LIN {X 0,Y 373.516,Z 952.695,A -85,B 0,C 180,E1 18425.825,E2 18425.825} C_VEL
LIN {X 0,Y 376.652,Z 940.388,A -85,B 0,C 180,E1 18422.322,E2 18422.322} C_VEL
LIN {X 0,Y 380.104,Z 927.885,A -85,B 0,C 180,E1 18419.319,E2 18419.319} C_VEL
LIN {X 0,Y 384.269,Z 913.225,A -85,B 0,C 180,E1 18416.347,E2 18416.347} C_VEL
LIN {X 0,Y 388.82,Z 897.706,A -85,B 0,C 180,E1 18413.653,E2 18413.653} C_VEL
LIN {X 0,Y 393.494,Z 881.198,A -85,B 0,C 180,E1 18411.233,E2 18411.233} C_VEL
LIN {X 0,Y 398.594,Z 862.696,A -85,B 0,C 180,E1 18408.917,E2 18408.917} C_VEL
LIN {X 0,Y 403.277,Z 844.718,A -85,B 0,C 180,E1 18407.02,E2 18407.02} C_VEL
LIN {X 0,Y 408.104,Z 824.554,A -85,B 0,C 180,E1 18405.227,E2 18405.227} C_VEL
LIN {X 0,Y 411.988,Z 806.631,A -85,B 0,C 180,E1 18403.886,E2 18403.886} C_VEL
LIN {X 0,Y 416.257,Z 784.1,A -85,B 0,C 180,E1 18402.494,E2 18402.494} C_VEL
LIN {X 0,Y 419.472,Z 764.172,A -85,B 0,C 180,E1 18401.502,E2 18401.502} C_VEL
LIN {X 0,Y 422.462,Z 740.832,A -85,B 0,C 180,E1 18400.598,E2 18400.598} C_VEL
LIN {X 0,Y 424.7,Z 718.024,A -85,B 0,C 180,E1 18399.95,E2 18399.95} C_VEL
LIN {X 0,Y 427.255,Z 666.6,A -85,B 0,C 180,E1 18398.953,E2 18398.953} C_VEL
LIN {X 0,Y 436.486,Z 468.995,A -85,B 0,C 180,E1 18395.218,E2 18395.218} C_VEL
LIN {X 0,Y 426.222,Z 453.887,A -85,B 0,C 180,E1 18392.733,E2 18392.733} C_VEL
LIN {X 0,Y 415.395,Z 439.157,A -85,B 0,C 180,E1 18389.805,E2 18389.805} C_VEL
LIN {X 0,Y 406.554,Z 427.967,A -85,B 0,C 180,E1 18387.103,E2 18387.103} C_VEL
LIN {X 0,Y 401.998,Z 422.413,A -85,B 0,C 180,E1 18385.565,E2 18385.565} C_VEL
LIN {X 0,Y 398.336,Z 417.839,A -85,B 0,C 180,E1 18384.23,E2 18384.23} C_VEL
LIN {X 0,Y 393.924,Z 412.857,A -85,B 0,C 180,E1 18382.511,E2 18382.511} C_VEL
LIN {X 0,Y 392.689,Z 411.071,A -85,B 0,C 180,E1 18381.981,E2 18381.981} C_VEL
LIN {X 0,Y 389.373,Z 407.904,A -85,B 0,C 180,E1 18380.558,E2 18380.558} C_VEL
LIN {X 0,Y 387.428,Z 404.914,A -85,B 0,C 180,E1 18379.603,E2 18379.603} C_VEL
LIN {X 0,Y 383.951,Z 402.051,A -85,B 0,C 180,E1 18377.896,E2 18377.896} C_VEL
LIN {X 0,Y 382.021,Z 398.482,A -85,B 0,C 180,E1 18376.733,E2 18376.733} C_VEL
LIN {X 0,Y 378.538,Z 396.352,A -85,B 0,C 180,E1 18374.689,E2 18374.689} C_VEL
LIN {X 0,Y 376.63,Z 393.429,A -85,B 0,C 180,E1 18373.276,E2 18373.276} C_VEL
LIN {X 0,Y 376.047,Z 391.834,A -85,B 0,C 180,E1 18372.75,E2 18372.75} C_VEL
LIN {X 0,Y 372.15,Z 389.796,A -85,B 0,C 180,E1 18369.433,E2 18369.433} C_VEL
LIN {X 0,Y 370.046,Z 386.524,A -85,B 0,C 180,E1 18366.594,E2 18366.594} C_VEL
LIN {X 0,Y 369.697,Z 384.985,A -85,B 0,C 180,E1 18365.639,E2 18365.639} C_VEL
LIN {X 0,Y 369.684,Z 384.983,A -85,B 0,C 180,E1 18361.705,E2 18361.705} C_VEL
LIN {X 0,Y 369.678,Z 384.981,A -85,B 0,C 180,E1 18357.675,E2 18357.675} C_VEL
LIN {X 0,Y 369.728,Z 385.142,A -85,B 0,C 180,E1 18354.608,E2 18354.608} C_VEL
LIN {X 0,Y 370.458,Z 387.543,A -85,B 0,C 180,E1 18353.18,E2 18353.18} C_VEL
LIN {X 0,Y 373.077,Z 390.581,A -85,B 0,C 180,E1 18350.124,E2 18350.124} C_VEL
LIN {X 0,Y 376.149,Z 392.051,A -85,B 0,C 180,E1 18347.645,E2 18347.645} C_VEL
LIN {X 0,Y 377.796,Z 395.551,A -85,B 0,C 180,E1 18346.299,E2 18346.299} C_VEL
LIN {X 0,Y 380.714,Z 397.973,A -85,B 0,C 180,E1 18344.462,E2 18344.462} C_VEL
LIN {X 0,Y 382.155,Z 398.748,A -85,B 0,C 180,E1 18343.665,E2 18343.665} C_VEL
LIN {X 0,Y 384.237,Z 402.413,A -85,B 0,C 180,E1 18342.431,E2 18342.431} C_VEL
LIN {X 0,Y 387.814,Z 405.39,A -85,B 0,C 180,E1 18340.692,E2 18340.692} C_VEL
LIN {X 0,Y 390.392,Z 409.19,A -85,B 0,C 180,E1 18339.459,E2 18339.459} C_VEL
LIN {X 0,Y 393.289,Z 411.748,A -85,B 0,C 180,E1 18338.252,E2 18338.252} C_VEL
LIN {X 0,Y 396.375,Z 415.904,A -85,B 0,C 180,E1 18336.984,E2 18336.984} C_VEL
LIN {X 0,Y 398.445,Z 418.003,A -85,B 0,C 180,E1 18336.21,E2 18336.21} C_VEL
LIN {X 0,Y 405.924,Z 427.773,A -85,B 0,C 180,E1 18333.563,E2 18333.563} C_VEL
LIN {X 0,Y 413.865,Z 438.738,A -85,B 0,C 180,E1 18331.068,E2 18331.068} C_VEL
LIN {X 0,Y 422.741,Z 451.748,A -85,B 0,C 180,E1 18328.566,E2 18328.566} C_VEL
LIN {X 0,Y 431.121,Z 464.861,A -85,B 0,C 180,E1 18326.418,E2 18326.418} C_VEL
LIN {X 0,Y 436.61,Z 474.131,A -85,B 0,C 180,E1 18325.098,E2 18325.098} C_VEL
LIN {X 0,Y 427.077,Z 679.523,A -85,B 0,C 180,E1 18321.22,E2 18321.22} C_VEL
LIN {X 0,Y 424.258,Z 738.023,A -85,B 0,C 180,E1 18320.092,E2 18320.092} C_VEL
LIN {X 0,Y 421.886,Z 761.213,A -85,B 0,C 180,E1 18319.459,E2 18319.459} C_VEL
LIN {X 0,Y 418.914,Z 783.591,A -85,B 0,C 180,E1 18318.636,E2 18318.636} C_VEL
LIN {X 0,Y 415.436,Z 804.583,A -85,B 0,C 180,E1 18317.629,E2 18317.629} C_VEL
LIN {X 0,Y 411.179,Z 826.892,A -85,B 0,C 180,E1 18316.297,E2 18316.297} C_VEL
LIN {X 0,Y 406.878,Z 846.732,A -85,B 0,C 180,E1 18314.845,E2 18314.845} C_VEL
LIN {X 0,Y 401.839,Z 867.94,A -85,B 0,C 180,E1 18312.976,E2 18312.976} C_VEL
LIN {X 0,Y 397.191,Z 886.217,A -85,B 0,C 180,E1 18311.068,E2 18311.068} C_VEL
LIN {X 0,Y 392.279,Z 904.4,A -85,B 0,C 180,E1 18308.825,E2 18308.825} C_VEL
LIN {X 0,Y 387.533,Z 921.911,A -85,B 0,C 180,E1 18306.303,E2 18306.303} C_VEL
LIN {X 0,Y 383.114,Z 937.825,A -85,B 0,C 180,E1 18303.589,E2 18303.589} C_VEL
LIN {X 0,Y 379.106,Z 952.905,A -85,B 0,C 180,E1 18300.595,E2 18300.595} C_VEL
LIN {X 0,Y 375.901,Z 965.517,A -85,B 0,C 180,E1 18297.658,E2 18297.658} C_VEL
LIN {X 0,Y 372.991,Z 978.095,A -85,B 0,C 180,E1 18294.211,E2 18294.211} C_VEL
LIN {X 0,Y 371.011,Z 987.984,A -85,B 0,C 180,E1 18291.002,E2 18291.002} C_VEL
LIN {X 0,Y 369.511,Z 996.933,A -85,B 0,C 180,E1 18287.477,E2 18287.477} C_VEL
LIN {X 0,Y 368.666,Z 1003.581,A -85,B 0,C 180,E1 18284.287,E2 18284.287} C_VEL
LIN {X 0,Y 368.17,Z 1009.216,A -85,B 0,C 180,E1 18280.799,E2 18280.799} C_VEL
LIN {X 0,Y 367.983,Z 1012.808,A -85,B 0,C 180,E1 18277.808,E2 18277.808} C_VEL
LIN {X 0,Y 367.925,Z 1015.554,A -85,B 0,C 180,E1 18274.364,E2 18274.364} C_VEL
LIN {X 0,Y 367.923,Z 1016.636,A -85,B 0,C 180,E1 18271.246,E2 18271.246} C_VEL
LIN {X 0,Y 367.927,Z 1016.566,A -85,B 0,C 180,E1 18268.288,E2 18268.288} C_VEL
LIN {X 0,Y 367.929,Z 1015.054,A -85,B 0,C 180,E1 18264.856,E2 18264.856} C_VEL
LIN {X 0,Y 368.017,Z 1012.314,A -85,B 0,C 180,E1 18261.722,E2 18261.722} C_VEL
LIN {X 0,Y 368.261,Z 1007.893,A -85,B 0,C 180,E1 18258.252,E2 18258.252} C_VEL
LIN {X 0,Y 368.84,Z 1002.025,A -85,B 0,C 180,E1 18254.918,E2 18254.918} C_VEL
LIN {X 0,Y 369.87,Z 994.748,A -85,B 0,C 180,E1 18251.564,E2 18251.564} C_VEL
LIN {X 0,Y 371.459,Z 985.641,A -85,B 0,C 180,E1 18248.198,E2 18248.198} C_VEL
LIN {X 0,Y 373.742,Z 974.864,A -85,B 0,C 180,E1 18244.83,E2 18244.83} C_VEL
LIN {X 0,Y 376.621,Z 962.624,A -85,B 0,C 180,E1 18241.631,E2 18241.631} C_VEL
LIN {X 0,Y 380.349,Z 948.091,A -85,B 0,C 180,E1 18238.399,E2 18238.399} C_VEL
LIN {X 0,Y 384.315,Z 933.523,A -85,B 0,C 180,E1 18235.633,E2 18235.633} C_VEL
LIN {X 0,Y 388.884,Z 916.777,A -85,B 0,C 180,E1 18232.926,E2 18232.926} C_VEL
LIN {X 0,Y 393.604,Z 899.717,A -85,B 0,C 180,E1 18230.555,E2 18230.555} C_VEL
LIN {X 0,Y 398.399,Z 881.4,A -85,B 0,C 180,E1 18228.407,E2 18228.407} C_VEL
LIN {X 0,Y 403.332,Z 861.809,A -85,B 0,C 180,E1 18226.443,E2 18226.443} C_VEL
LIN {X 0,Y 407.884,Z 842.145,A -85,B 0,C 180,E1 18224.8,E2 18224.8} C_VEL
LIN {X 0,Y 412.556,Z 819.977,A -85,B 0,C 180,E1 18223.265,E2 18223.265} C_VEL
LIN {X 0,Y 416.124,Z 800.624,A -85,B 0,C 180,E1 18222.169,E2 18222.169} C_VEL
LIN {X 0,Y 419.768,Z 777.421,A -85,B 0,C 180,E1 18221.121,E2 18221.121} C_VEL
LIN {X 0,Y 422.274,Z 757.737,A -85,B 0,C 180,E1 18220.438,E2 18220.438} C_VEL
LIN {X 0,Y 424.553,Z 732.637,A -85,B 0,C 180,E1 18219.8,E2 18219.8} C_VEL
LIN {X 0,Y 433.641,Z 535.185,A -85,B 0,C 180,E1 18216.062,E2 18216.062} C_VEL
LIN {X 0,Y 436.481,Z 473.671,A -85,B 0,C 180,E1 18214.879,E2 18214.879} C_VEL
LIN {X 0,Y 426.008,Z 456.76,A -85,B 0,C 180,E1 18212.312,E2 18212.312} C_VEL
LIN {X 0,Y 415.5,Z 441.08,A -85,B 0,C 180,E1 18209.439,E2 18209.439} C_VEL
LIN {X 0,Y 407.607,Z 430.178,A -85,B 0,C 180,E1 18207.027,E2 18207.027} C_VEL
LIN {X 0,Y 403.606,Z 424.766,A -85,B 0,C 180,E1 18205.691,E2 18205.691} C_VEL
LIN {X 0,Y 397.54,Z 416.927,A -85,B 0,C 180,E1 18203.493,E2 18203.493} C_VEL
LIN {X 0,Y 394.055,Z 413.056,A -85,B 0,C 180,E1 18202.135,E2 18202.135} C_VEL
LIN {X 0,Y 392.767,Z 411.133,A -85,B 0,C 180,E1 18201.583,E2 18201.583} C_VEL
LIN {X 0,Y 389.194,Z 407.75,A -85,B 0,C 180,E1 18200.057,E2 18200.057} C_VEL
LIN {X 0,Y 387.321,Z 404.835,A -85,B 0,C 180,E1 18199.138,E2 18199.138} C_VEL
LIN {X 0,Y 384.105,Z 402.262,A -85,B 0,C 180,E1 18197.575,E2 18197.575} C_VEL
LIN {X 0,Y 381.889,Z 398.463,A -85,B 0,C 180,E1 18196.269,E2 18196.269} C_VEL
LIN {X 0,Y 378.287,Z 396.166,A -85,B 0,C 180,E1 18194.151,E2 18194.151} C_VEL
LIN {X 0,Y 376.466,Z 393.014,A -85,B 0,C 180,E1 18192.774,E2 18192.774} C_VEL
LIN {X 0,Y 376.101,Z 391.867,A -85,B 0,C 180,E1 18192.435,E2 18192.435} C_VEL
LIN {X 0,Y 372.429,Z 390.055,A -85,B 0,C 180,E1 18189.425,E2 18189.425} C_VEL
LIN {X 0,Y 370.155,Z 386.892,A -85,B 0,C 180,E1 18186.606,E2 18186.606} C_VEL
LIN {X 0,Y 369.687,Z 384.981,A -85,B 0,C 180,E1 18185.587,E2 18185.587} C_VEL
LIN {X 0,Y 369.689,Z 384.981,A -85,B 0,C 180,E1 18181.549,E2 18181.549} C_VEL
LIN {X 0,Y 369.681,Z 384.984,A -85,B 0,C 180,E1 18177.675,E2 18177.675} C_VEL
LIN {X 0,Y 369.686,Z 385.014,A -85,B 0,C 180,E1 18173.789,E2 18173.789} C_VEL
LIN {X 0,Y 370.975,Z 388.444,A -85,B 0,C 180,E1 18171.631,E2 18171.631} C_VEL
LIN {X 0,Y 374.173,Z 391.196,A -85,B 0,C 180,E1 18168.439,E2 18168.439} C_VEL
LIN {X 0,Y 376.158,Z 392.014,A -85,B 0,C 180,E1 18166.942,E2 18166.942} C_VEL
LIN {X 0,Y 377.412,Z 395.001,A -85,B 0,C 180,E1 18165.893,E2 18165.893} C_VEL
LIN {X 0,Y 380.397,Z 397.79,A -85,B 0,C 180,E1 18163.979,E2 18163.979} C_VEL
LIN {X 0,Y 382.105,Z 398.687,A -85,B 0,C 180,E1 18163.036,E2 18163.036} C_VEL
LIN {X 0,Y 384.066,Z 402.206,A -85,B 0,C 180,E1 18161.874,E2 18161.874} C_VEL
LIN {X 0,Y 387.875,Z 405.412,A -85,B 0,C 180,E1 18160.028,E2 18160.028} C_VEL
LIN {X 0,Y 390.547,Z 409.351,A -85,B 0,C 180,E1 18158.761,E2 18158.761} C_VEL
LIN {X 0,Y 393.213,Z 411.691,A -85,B 0,C 180,E1 18157.657,E2 18157.657} C_VEL
LIN {X 0,Y 396.4,Z 415.938,A -85,B 0,C 180,E1 18156.356,E2 18156.356} C_VEL
LIN {X 0,Y 398.299,Z 417.824,A -85,B 0,C 180,E1 18155.649,E2 18155.649} C_VEL
LIN {X 0,Y 401.875,Z 422.318,A -85,B 0,C 180,E1 18154.347,E2 18154.347} C_VEL
LIN {X 0,Y 403.594,Z 424.397,A -85,B 0,C 180,E1 18153.755,E2 18153.755} C_VEL
LIN {X 0,Y 408.142,Z 430.056,A -85,B 0,C 180,E1 18152.26,E2 18152.26} C_VEL
LIN {X 0,Y 413.122,Z 436.484,A -85,B 0,C 180,E1 18150.732,E2 18150.732} C_VEL
LIN {X 0,Y 419.587,Z 444.835,A -85,B 0,C 180,E1 18148.902,E2 18148.902} C_VEL
LIN {X 0,Y 429.926,Z 459.317,A -85,B 0,C 180,E1 18146.232,E2 18146.232} C_VEL
LIN {X 0,Y 436.465,Z 469.171,A -85,B 0,C 180,E1 18144.678,E2 18144.678} C_VEL
LIN {X 0,Y 426.653,Z 679.212,A -85,B 0,C 180,E1 18140.716,E2 18140.716} C_VEL
LIN {X 0,Y 424.59,Z 718.849,A -85,B 0,C 180,E1 18139.935,E2 18139.935} C_VEL
LIN {X 0,Y 422.399,Z 741.121,A -85,B 0,C 180,E1 18139.298,E2 18139.298} C_VEL
LIN {X 0,Y 419.325,Z 764.94,A -85,B 0,C 180,E1 18138.368,E2 18138.368} C_VEL
LIN {X 0,Y 416.219,Z 784.161,A -85,B 0,C 180,E1 18137.408,E2 18137.408} C_VEL
LIN {X 0,Y 411.978,Z 806.574,A -85,B 0,C 180,E1 18136.024,E2 18136.024} C_VEL
LIN {X 0,Y 408.075,Z 824.581,A -85,B 0,C 180,E1 18134.677,E2 18134.677} C_VEL
LIN {X 0,Y 403.062,Z 845.452,A -85,B 0,C 180,E1 18132.814,E2 18132.814} C_VEL
LIN {X 0,Y 398.238,Z 864.016,A -85,B 0,C 180,E1 18130.841,E2 18130.841} C_VEL
LIN {X 0,Y 393.344,Z 881.688,A -85,B 0,C 180,E1 18128.606,E2 18128.606} C_VEL
LIN {X 0,Y 388.676,Z 898.193,A -85,B 0,C 180,E1 18126.179,E2 18126.179} C_VEL
LIN {X 0,Y 384.149,Z 913.628,A -85,B 0,C 180,E1 18123.485,E2 18123.485} C_VEL
LIN {X 0,Y 380.002,Z 928.214,A -85,B 0,C 180,E1 18120.514,E2 18120.514} C_VEL
LIN {X 0,Y 378.162,Z 934.959,A -85,B 0,C 180,E1 18118.963,E2 18118.963} C_VEL
LIN {X 0,Y 376.147,Z 939.177,A -85,B 0,C 180,E1 18118.021,E2 18118.021} C_VEL
LIN {X 0,Y 367.506,Z 949.935,A -85,B 0,C 180,E1 18115.527,E2 18115.527} C_VEL
LIN {X 0,Y 366.002,Z 952.956,A -85,B 0,C 180,E1 18114.63,E2 18114.63} C_VEL
LIN {X 0,Y 363.682,Z 962.63,A -85,B 0,C 180,E1 18111.276,E2 18111.276} C_VEL
LIN {X 0,Y 362.005,Z 970.702,A -85,B 0,C 180,E1 18107.851,E2 18107.851} C_VEL
LIN {X 0,Y 360.935,Z 977.299,A -85,B 0,C 180,E1 18104.435,E2 18104.435} C_VEL
LIN {X 0,Y 360.306,Z 982.537,A -85,B 0,C 180,E1 18100.875,E2 18100.875} C_VEL
LIN {X 0,Y 360.034,Z 986.031,A -85,B 0,C 180,E1 18097.659,E2 18097.659} C_VEL
LIN {X 0,Y 359.946,Z 988.516,A -85,B 0,C 180,E1 18093.981,E2 18093.981} C_VEL
LIN {X 0,Y 359.922,Z 989.386,A -85,B 0,C 180,E1 18090.954,E2 18090.954} C_VEL
LIN {X 0,Y 359.937,Z 989.147,A -85,B 0,C 180,E1 18087.452,E2 18087.452} C_VEL
LIN {X 0,Y 359.975,Z 987.462,A -85,B 0,C 180,E1 18084.102,E2 18084.102} C_VEL
LIN {X 0,Y 360.165,Z 984.418,A -85,B 0,C 180,E1 18080.574,E2 18080.574} C_VEL
LIN {X 0,Y 360.615,Z 979.736,A -85,B 0,C 180,E1 18077.023,E2 18077.023} C_VEL
LIN {X 0,Y 361.527,Z 973.629,A -85,B 0,C 180,E1 18073.451,E2 18073.451} C_VEL
LIN {X 0,Y 363.012,Z 965.68,A -85,B 0,C 180,E1 18069.863,E2 18069.863} C_VEL
LIN {X 0,Y 365.253,Z 956.02,A -85,B 0,C 180,E1 18066.274,E2 18066.274} C_VEL
LIN {X 0,Y 367.859,Z 945.995,A -85,B 0,C 180,E1 18063.182,E2 18063.182} C_VEL
LIN {X 0,Y 371.648,Z 932.713,A -85,B 0,C 180,E1 18059.723,E2 18059.723} C_VEL
LIN {X 0,Y 375.474,Z 919.99,A -85,B 0,C 180,E1 18056.918,E2 18056.918} C_VEL
LIN {X 0,Y 380.055,Z 904.898,A -85,B 0,C 180,E1 18054.083,E2 18054.083} C_VEL
LIN {X 0,Y 384.914,Z 889.023,A -85,B 0,C 180,E1 18051.533,E2 18051.533} C_VEL
LIN {X 0,Y 389.998,Z 871.654,A -85,B 0,C 180,E1 18049.18,E2 18049.18} C_VEL
LIN {X 0,Y 395.062,Z 853.737,A -85,B 0,C 180,E1 18047.099,E2 18047.099} C_VEL
LIN {X 0,Y 400.045,Z 834.352,A -85,B 0,C 180,E1 18045.22,E2 18045.22} C_VEL
LIN {X 0,Y 404.945,Z 813.698,A -85,B 0,C 180,E1 18043.542,E2 18043.542} C_VEL
LIN {X 0,Y 408.969,Z 794.385,A -85,B 0,C 180,E1 18042.247,E2 18042.247} C_VEL
LIN {X 0,Y 412.949,Z 772.361,A -85,B 0,C 180,E1 18041.039,E2 18041.039} C_VEL
LIN {X 0,Y 415.872,Z 752.629,A -85,B 0,C 180,E1 18040.18,E2 18040.18} C_VEL
LIN {X 0,Y 418.6,Z 729.318,A -85,B 0,C 180,E1 18039.403,E2 18039.403} C_VEL
LIN {X 0,Y 420.287,Z 707.78,A -85,B 0,C 180,E1 18038.891,E2 18038.891} C_VEL
LIN {X 0,Y 430.38,Z 500.127,A -85,B 0,C 180,E1 18034.943,E2 18034.943} C_VEL
LIN {X 0,Y 431.677,Z 473.073,A -85,B 0,C 180,E1 18034.413,E2 18034.413} C_VEL
LIN {X 0,Y 422.102,Z 459.129,A -85,B 0,C 180,E1 18032.01,E2 18032.01} C_VEL
LIN {X 0,Y 412.697,Z 446.062,A -85,B 0,C 180,E1 18029.381,E2 18029.381} C_VEL
LIN {X 0,Y 404.001,Z 434.917,A -85,B 0,C 180,E1 18026.653,E2 18026.653} C_VEL
LIN {X 0,Y 399.715,Z 429.598,A -85,B 0,C 180,E1 18025.166,E2 18025.166} C_VEL
LIN {X 0,Y 395.232,Z 424.08,A -85,B 0,C 180,E1 18023.481,E2 18023.481} C_VEL
LIN {X 0,Y 391.692,Z 419.829,A -85,B 0,C 180,E1 18022.04,E2 18022.04} C_VEL
LIN {X 0,Y 390.567,Z 418.418,A -85,B 0,C 180,E1 18021.553,E2 18021.553} C_VEL
LIN {X 0,Y 387.275,Z 414.949,A -85,B 0,C 180,E1 18020.083,E2 18020.083} C_VEL
LIN {X 0,Y 385.875,Z 412.632,A -85,B 0,C 180,E1 18019.37,E2 18019.37} C_VEL
LIN {X 0,Y 382.317,Z 409.595,A -85,B 0,C 180,E1 18017.582,E2 18017.582} C_VEL
LIN {X 0,Y 380.274,Z 406.175,A -85,B 0,C 180,E1 18016.34,E2 18016.34} C_VEL
LIN {X 0,Y 376.699,Z 403.582,A -85,B 0,C 180,E1 18014.134,E2 18014.134} C_VEL
LIN {X 0,Y 374.92,Z 400.343,A -85,B 0,C 180,E1 18012.71,E2 18012.71} C_VEL
LIN {X 0,Y 374.677,Z 399.689,A -85,B 0,C 180,E1 18012.484,E2 18012.484} C_VEL
LIN {X 0,Y 370.899,Z 397.528,A -85,B 0,C 180,E1 18009.152,E2 18009.152} C_VEL
LIN {X 0,Y 368.891,Z 394.216,A -85,B 0,C 180,E1 18006.303,E2 18006.303} C_VEL
LIN {X 0,Y 368.513,Z 392.892,A -85,B 0,C 180,E1 18005.45,E2 18005.45} C_VEL
LIN {X 0,Y 367.439,Z 392.659,A -85,B 0,C 180,E1 17997.505,E2 17997.505} C_VEL
LIN {X 0,Y 368.629,Z 393.15,A -85,B 0,C 180,E1 17994.787,E2 17994.787} C_VEL
LIN {X 0,Y 369.683,Z 395.969,A -85,B 0,C 180,E1 17992.853,E2 17992.853} C_VEL
LIN {X 0,Y 372.612,Z 398.888,A -85,B 0,C 180,E1 17989.643,E2 17989.643} C_VEL
LIN {X 0,Y 374.769,Z 399.953,A -85,B 0,C 180,E1 17987.911,E2 17987.911} C_VEL
LIN {X 0,Y 376.71,Z 403.645,A -85,B 0,C 180,E1 17986.337,E2 17986.337} C_VEL
LIN {X 0,Y 380.027,Z 406.102,A -85,B 0,C 180,E1 17984.277,E2 17984.277} C_VEL
LIN {X 0,Y 380.708,Z 406.819,A -85,B 0,C 180,E1 17983.875,E2 17983.875} C_VEL
LIN {X 0,Y 383.131,Z 410.56,A -85,B 0,C 180,E1 17982.457,E2 17982.457} C_VEL
LIN {X 0,Y 386.091,Z 413.082,A -85,B 0,C 180,E1 17980.995,E2 17980.995} C_VEL
LIN {X 0,Y 388.957,Z 417.048,A -85,B 0,C 180,E1 17979.616,E2 17979.616} C_VEL
LIN {X 0,Y 391.403,Z 419.31,A -85,B 0,C 180,E1 17978.574,E2 17978.574} C_VEL
LIN {X 0,Y 394.717,Z 423.618,A -85,B 0,C 180,E1 17977.197,E2 17977.197} C_VEL
LIN {X 0,Y 396.48,Z 425.573,A -85,B 0,C 180,E1 17976.519,E2 17976.519} C_VEL
LIN {X 0,Y 403.385,Z 434.649,A -85,B 0,C 180,E1 17974.017,E2 17974.017} C_VEL
LIN {X 0,Y 411.707,Z 446.397,A -85,B 0,C 180,E1 17971.338,E2 17971.338} C_VEL
LIN {X 0,Y 420.037,Z 458.848,A -85,B 0,C 180,E1 17968.939,E2 17968.939} C_VEL
LIN {X 0,Y 428.31,Z 472.015,A -85,B 0,C 180,E1 17966.77,E2 17966.77} C_VEL
LIN {X 0,Y 431.837,Z 478.104,A -85,B 0,C 180,E1 17965.893,E2 17965.893} C_VEL
LIN {X 0,Y 421.794,Z 685.475,A -85,B 0,C 180,E1 17961.954,E2 17961.954} C_VEL
LIN {X 0,Y 419.118,Z 738.028,A -85,B 0,C 180,E1 17960.929,E2 17960.929} C_VEL
LIN {X 0,Y 416.677,Z 761.053,A -85,B 0,C 180,E1 17960.297,E2 17960.297} C_VEL
LIN {X 0,Y 413.691,Z 782.846,A -85,B 0,C 180,E1 17959.497,E2 17959.497} C_VEL
LIN {X 0,Y 410.003,Z 804.285,A -85,B 0,C 180,E1 17958.468,E2 17958.468} C_VEL
LIN {X 0,Y 405.649,Z 826.242,A -85,B 0,C 180,E1 17957.156,E2 17957.156} C_VEL
LIN {X 0,Y 401.087,Z 846.428,A -85,B 0,C 180,E1 17955.674,E2 17955.674} C_VEL
LIN {X 0,Y 395.823,Z 867.634,A -85,B 0,C 180,E1 17953.793,E2 17953.793} C_VEL
LIN {X 0,Y 390.967,Z 885.909,A -85,B 0,C 180,E1 17951.867,E2 17951.867} C_VEL
LIN {X 0,Y 385.818,Z 904.09,A -85,B 0,C 180,E1 17949.602,E2 17949.602} C_VEL
LIN {X 0,Y 380.953,Z 921.104,A -85,B 0,C 180,E1 17947.128,E2 17947.128} C_VEL
LIN {X 0,Y 376.408,Z 936.653,A -85,B 0,C 180,E1 17944.454,E2 17944.454} C_VEL
LIN {X 0,Y 372.312,Z 951.164,A -85,B 0,C 180,E1 17941.576,E2 17941.576} C_VEL
LIN {X 0,Y 368.745,Z 964.252,A -85,B 0,C 180,E1 17938.501,E2 17938.501} C_VEL
LIN {X 0,Y 365.655,Z 976.73,A -85,B 0,C 180,E1 17935.074,E2 17935.074} C_VEL
LIN {X 0,Y 363.454,Z 986.733,A -85,B 0,C 180,E1 17931.799,E2 17931.799} C_VEL
LIN {X 0,Y 361.704,Z 996.275,A -85,B 0,C 180,E1 17928.027,E2 17928.027} C_VEL
LIN {X 0,Y 360.765,Z 1002.962,A -85,B 0,C 180,E1 17924.771,E2 17924.771} C_VEL
LIN {X 0,Y 360.192,Z 1008.911,A -85,B 0,C 180,E1 17921.042,E2 17921.042} C_VEL
LIN {X 0,Y 360.001,Z 1012.505,A -85,B 0,C 180,E1 17917.982,E2 17917.982} C_VEL
LIN {X 0,Y 359.927,Z 1015.253,A -85,B 0,C 180,E1 17914.461,E2 17914.461} C_VEL
LIN {X 0,Y 359.929,Z 1016.336,A -85,B 0,C 180,E1 17911.274,E2 17911.274} C_VEL
LIN {X 0,Y 359.933,Z 1016.266,A -85,B 0,C 180,E1 17908.25,E2 17908.25} C_VEL
LIN {X 0,Y 359.933,Z 1014.753,A -85,B 0,C 180,E1 17904.741,E2 17904.741} C_VEL
LIN {X 0,Y 360.026,Z 1012.011,A -85,B 0,C 180,E1 17901.537,E2 17901.537} C_VEL
LIN {X 0,Y 360.296,Z 1007.588,A -85,B 0,C 180,E1 17897.989,E2 17897.989} C_VEL
LIN {X 0,Y 360.924,Z 1001.718,A -85,B 0,C 180,E1 17894.579,E2 17894.579} C_VEL
LIN {X 0,Y 362.036,Z 994.438,A -85,B 0,C 180,E1 17891.151,E2 17891.151} C_VEL
LIN {X 0,Y 363.733,Z 985.328,A -85,B 0,C 180,E1 17887.71,E2 17887.71} C_VEL
LIN {X 0,Y 366.18,Z 974.549,A -85,B 0,C 180,E1 17884.272,E2 17884.272} C_VEL
LIN {X 0,Y 369.089,Z 962.957,A -85,B 0,C 180,E1 17881.175,E2 17881.175} C_VEL
LIN {X 0,Y 372.999,Z 948.601,A -85,B 0,C 180,E1 17877.893,E2 17877.893} C_VEL
LIN {X 0,Y 377.159,Z 934.065,A -85,B 0,C 180,E1 17875.072,E2 17875.072} C_VEL
LIN {X 0,Y 382.095,Z 916.975,A -85,B 0,C 180,E1 17872.248,E2 17872.248} C_VEL
LIN {X 0,Y 387.24,Z 899.266,A -85,B 0,C 180,E1 17869.753,E2 17869.753} C_VEL
LIN {X 0,Y 392.391,Z 880.467,A -85,B 0,C 180,E1 17867.533,E2 17867.533} C_VEL
LIN {X 0,Y 397.789,Z 859.857,A -85,B 0,C 180,E1 17865.477,E2 17865.477} C_VEL
LIN {X 0,Y 402.408,Z 840.737,A -85,B 0,C 180,E1 17863.886,E2 17863.886} C_VEL
LIN {X 0,Y 407.231,Z 818.525,A -85,B 0,C 180,E1 17862.359,E2 17862.359} C_VEL
LIN {X 0,Y 410.955,Z 799.02,A -85,B 0,C 180,E1 17861.261,E2 17861.261} C_VEL
LIN {X 0,Y 414.658,Z 775.898,A -85,B 0,C 180,E1 17860.231,E2 17860.231} C_VEL
LIN {X 0,Y 417.305,Z 755.69,A -85,B 0,C 180,E1 17859.541,E2 17859.541} C_VEL
LIN {X 0,Y 419.494,Z 731.564,A -85,B 0,C 180,E1 17858.939,E2 17858.939} C_VEL
LIN {X 0,Y 429.116,Z 531.431,A -85,B 0,C 180,E1 17855.127,E2 17855.127} C_VEL
LIN {X 0,Y 431.715,Z 477.737,A -85,B 0,C 180,E1 17854.088,E2 17854.088} C_VEL
LIN {X 0,Y 421.551,Z 461.203,A -85,B 0,C 180,E1 17851.493,E2 17851.493} C_VEL
LIN {X 0,Y 412.261,Z 447.228,A -85,B 0,C 180,E1 17848.857,E2 17848.857} C_VEL
LIN {X 0,Y 404.835,Z 436.798,A -85,B 0,C 180,E1 17846.513,E2 17846.513} C_VEL
LIN {X 0,Y 399.633,Z 429.56,A -85,B 0,C 180,E1 17844.697,E2 17844.697} C_VEL
LIN {X 0,Y 395.324,Z 424.172,A -85,B 0,C 180,E1 17843.08,E2 17843.08} C_VEL
LIN {X 0,Y 391.761,Z 419.943,A -85,B 0,C 180,E1 17841.641,E2 17841.641} C_VEL
LIN {X 0,Y 390.636,Z 418.478,A -85,B 0,C 180,E1 17841.155,E2 17841.155} C_VEL
LIN {X 0,Y 387.092,Z 414.794,A -85,B 0,C 180,E1 17839.581,E2 17839.581} C_VEL
LIN {X 0,Y 385.764,Z 412.555,A -85,B 0,C 180,E1 17838.904,E2 17838.904} C_VEL
LIN {X 0,Y 382.462,Z 409.803,A -85,B 0,C 180,E1 17837.26,E2 17837.26} C_VEL
LIN {X 0,Y 380.406,Z 406.247,A -85,B 0,C 180,E1 17836.02,E2 17836.02} C_VEL
LIN {X 0,Y 376.77,Z 403.73,A -85,B 0,C 180,E1 17833.818,E2 17833.818} C_VEL
LIN {X 0,Y 374.875,Z 400.268,A -85,B 0,C 180,E1 17832.32,E2 17832.32} C_VEL
LIN {X 0,Y 374.517,Z 399.654,A -85,B 0,C 180,E1 17832.019,E2 17832.019} C_VEL
LIN {X 0,Y 370.868,Z 397.533,A -85,B 0,C 180,E1 17828.839,E2 17828.839} C_VEL
LIN {X 0,Y 368.809,Z 394.077,A -85,B 0,C 180,E1 17825.991,E2 17825.991} C_VEL
LIN {X 0,Y 368.49,Z 392.886,A -85,B 0,C 180,E1 17825.293,E2 17825.293} C_VEL
LIN {X 0,Y 367.099,Z 392.552,A -85,B 0,C 180,E1 17817.346,E2 17817.346} C_VEL
LIN {X 0,Y 368.597,Z 393.096,A -85,B 0,C 180,E1 17813.927,E2 17813.927} C_VEL
LIN {X 0,Y 369.997,Z 396.496,A -85,B 0,C 180,E1 17811.609,E2 17811.609} C_VEL
LIN {X 0,Y 373.214,Z 399.17,A -85,B 0,C 180,E1 17808.408,E2 17808.408} C_VEL
LIN {X 0,Y 374.767,Z 399.982,A -85,B 0,C 180,E1 17807.206,E2 17807.206} C_VEL
LIN {X 0,Y 376.427,Z 403.266,A -85,B 0,C 180,E1 17805.855,E2 17805.855} C_VEL
LIN {X 0,Y 379.708,Z 405.938,A -85,B 0,C 180,E1 17803.792,E2 17803.792} C_VEL
LIN {X 0,Y 380.598,Z 406.663,A -85,B 0,C 180,E1 17803.282,E2 17803.282} C_VEL
LIN {X 0,Y 382.961,Z 410.366,A -85,B 0,C 180,E1 17801.899,E2 17801.899} C_VEL
LIN {X 0,Y 386.151,Z 413.104,A -85,B 0,C 180,E1 17800.329,E2 17800.329} C_VEL
LIN {X 0,Y 389.112,Z 417.215,A -85,B 0,C 180,E1 17798.915,E2 17798.915} C_VEL
LIN {X 0,Y 391.327,Z 419.263,A -85,B 0,C 180,E1 17797.978,E2 17797.978} C_VEL
LIN {X 0,Y 394.742,Z 423.653,A -85,B 0,C 180,E1 17796.567,E2 17796.567} C_VEL
LIN {X 0,Y 396.336,Z 425.403,A -85,B 0,C 180,E1 17795.957,E2 17795.957} C_VEL
LIN {X 0,Y 400.166,Z 430.042,A -85,B 0,C 180,E1 17794.547,E2 17794.547} C_VEL
LIN {X 0,Y 406.056,Z 437.638,A -85,B 0,C 180,E1 17792.543,E2 17792.543} C_VEL
LIN {X 0,Y 413.233,Z 446.849,A -85,B 0,C 180,E1 17790.343,E2 17790.343} C_VEL
LIN {X 0,Y 423.624,Z 461.258,A -85,B 0,C 180,E1 17787.483,E2 17787.483} C_VEL
LIN {X 0,Y 431.69,Z 473.367,A -85,B 0,C 180,E1 17785.47,E2 17785.47} C_VEL
LIN {X 0,Y 421.503,Z 682.31,A -85,B 0,C 180,E1 17781.505,E2 17781.505} C_VEL
LIN {X 0,Y 419.454,Z 719.491,A -85,B 0,C 180,E1 17780.763,E2 17780.763} C_VEL
LIN {X 0,Y 417.186,Z 741.696,A -85,B 0,C 180,E1 17780.124,E2 17780.124} C_VEL
LIN {X 0,Y 414.028,Z 765.252,A -85,B 0,C 180,E1 17779.2,E2 17779.2} C_VEL
LIN {X 0,Y 410.804,Z 784.472,A -85,B 0,C 180,E1 17778.236,E2 17778.236} C_VEL
LIN {X 0,Y 406.411,Z 806.844,A -85,B 0,C 180,E1 17776.847,E2 17776.847} C_VEL
LIN {X 0,Y 402.341,Z 824.892,A -85,B 0,C 180,E1 17775.491,E2 17775.491} C_VEL
LIN {X 0,Y 397.123,Z 845.763,A -85,B 0,C 180,E1 17773.613,E2 17773.613} C_VEL
LIN {X 0,Y 392.198,Z 863.898,A -85,B 0,C 180,E1 17771.671,E2 17771.671} C_VEL
LIN {X 0,Y 386.966,Z 881.946,A -85,B 0,C 180,E1 17769.374,E2 17769.374} C_VEL
LIN {X 0,Y 382.053,Z 898.506,A -85,B 0,C 180,E1 17766.909,E2 17766.909} C_VEL
LIN {X 0,Y 377.281,Z 913.942,A -85,B 0,C 180,E1 17764.178,E2 17764.178} C_VEL
LIN {X 0,Y 372.899,Z 928.527,A -85,B 0,C 180,E1 17761.16,E2 17761.16} C_VEL
LIN {X 0,Y 369.425,Z 940.375,A -85,B 0,C 180,E1 17758.267,E2 17758.267} C_VEL
LIN {X 0,Y 366.002,Z 952.956,A -85,B 0,C 180,E1 17754.63,E2 17754.63} C_VEL
LIN {X 0,Y 364.194,Z 956.478,A -85,B 0,C 180,E1 17753.573,E2 17753.573} C_VEL
LIN {X 0,Y 356.173,Z 965.242,A -85,B 0,C 180,E1 17750.77,E2 17750.77} C_VEL
LIN {X 0,Y 354.931,Z 967.661,A -85,B 0,C 180,E1 17749.794,E2 17749.794} C_VEL
LIN {X 0,Y 353.382,Z 975.545,A -85,B 0,C 180,E1 17745.927,E2 17745.927} C_VEL
LIN {X 0,Y 352.558,Z 981.141,A -85,B 0,C 180,E1 17742.445,E2 17742.445} C_VEL
LIN {X 0,Y 352.129,Z 985.56,A -85,B 0,C 180,E1 17738.654,E2 17738.654} C_VEL
LIN {X 0,Y 351.974,Z 988.251,A -85,B 0,C 180,E1 17735.215,E2 17735.215} C_VEL
LIN {X 0,Y 351.94,Z 989.599,A -85,B 0,C 180,E1 17731.627,E2 17731.627} C_VEL
LIN {X 0,Y 351.94,Z 989.633,A -85,B 0,C 180,E1 17728.535,E2 17728.535} C_VEL
LIN {X 0,Y 351.967,Z 988.423,A -85,B 0,C 180,E1 17724.948,E2 17724.948} C_VEL
LIN {X 0,Y 352.113,Z 985.8,A -85,B 0,C 180,E1 17721.509,E2 17721.509} C_VEL
LIN {X 0,Y 352.482,Z 981.751,A -85,B 0,C 180,E1 17717.884,E2 17717.884} C_VEL
LIN {X 0,Y 353.317,Z 975.917,A -85,B 0,C 180,E1 17714.191,E2 17714.191} C_VEL
LIN {X 0,Y 354.711,Z 968.75,A -85,B 0,C 180,E1 17710.574,E2 17710.574} C_VEL
LIN {X 0,Y 356.723,Z 960.04,A -85,B 0,C 180,E1 17707.073,E2 17707.073} C_VEL
LIN {X 0,Y 359.694,Z 949.108,A -85,B 0,C 180,E1 17703.417,E2 17703.417} C_VEL
LIN {X 0,Y 363.029,Z 937.893,A -85,B 0,C 180,E1 17700.284,E2 17700.284} C_VEL
LIN {X 0,Y 367.335,Z 924.081,A -85,B 0,C 180,E1 17697.021,E2 17697.021} C_VEL
LIN {X 0,Y 372.003,Z 909.683,A -85,B 0,C 180,E1 17694.135,E2 17694.135} C_VEL
LIN {X 0,Y 377.033,Z 893.823,A -85,B 0,C 180,E1 17691.455,E2 17691.455} C_VEL
LIN {X 0,Y 382.415,Z 876.762,A -85,B 0,C 180,E1 17688.99,E2 17688.99} C_VEL
LIN {X 0,Y 387.558,Z 859.34,A -85,B 0,C 180,E1 17686.874,E2 17686.874} C_VEL
LIN {X 0,Y 392.932,Z 840.041,A -85,B 0,C 180,E1 17684.879,E2 17684.879} C_VEL
LIN {X 0,Y 397.589,Z 821.581,A -85,B 0,C 180,E1 17683.284,E2 17683.284} C_VEL
LIN {X 0,Y 402.536,Z 799.743,A -85,B 0,C 180,E1 17681.714,E2 17681.714} C_VEL
LIN {X 0,Y 406.474,Z 779.583,A -85,B 0,C 180,E1 17680.535,E2 17680.535} C_VEL
LIN {X 0,Y 410.223,Z 756.48,A -85,B 0,C 180,E1 17679.464,E2 17679.464} C_VEL
LIN {X 0,Y 413.031,Z 734.685,A -85,B 0,C 180,E1 17678.69,E2 17678.69} C_VEL
LIN {X 0,Y 415.08,Z 711.516,A -85,B 0,C 180,E1 17678.104,E2 17678.104} C_VEL
LIN {X 0,Y 425.379,Z 509.262,A -85,B 0,C 180,E1 17674.229,E2 17674.229} C_VEL
LIN {X 0,Y 426.939,Z 477.309,A -85,B 0,C 180,E1 17673.592,E2 17673.592} C_VEL
LIN {X 0,Y 418.038,Z 464.242,A -85,B 0,C 180,E1 17671.267,E2 17671.267} C_VEL
LIN {X 0,Y 409.809,Z 452.713,A -85,B 0,C 180,E1 17668.887,E2 17668.887} C_VEL
LIN {X 0,Y 401.571,Z 441.963,A -85,B 0,C 180,E1 17666.229,E2 17666.229} C_VEL
LIN {X 0,Y 397.429,Z 436.751,A -85,B 0,C 180,E1 17664.754,E2 17664.754} C_VEL
LIN {X 0,Y 393.224,Z 431.468,A -85,B 0,C 180,E1 17663.132,E2 17663.132} C_VEL
LIN {X 0,Y 389.59,Z 426.973,A -85,B 0,C 180,E1 17661.61,E2 17661.61} C_VEL
LIN {X 0,Y 387.511,Z 424.871,A -85,B 0,C 180,E1 17660.701,E2 17660.701} C_VEL
LIN {X 0,Y 384.382,Z 420.589,A -85,B 0,C 180,E1 17659.172,E2 17659.172} C_VEL
LIN {X 0,Y 380.32,Z 416.615,A -85,B 0,C 180,E1 17657.046,E2 17657.046} C_VEL
LIN {X 0,Y 378.807,Z 413.946,A -85,B 0,C 180,E1 17656.09,E2 17656.09} C_VEL
LIN {X 0,Y 375.205,Z 411.146,A -85,B 0,C 180,E1 17653.798,E2 17653.798} C_VEL
LIN {X 0,Y 373.399,Z 407.718,A -85,B 0,C 180,E1 17652.291,E2 17652.291} C_VEL
LIN {X 0,Y 369.269,Z 404.843,A -85,B 0,C 180,E1 17648.408,E2 17648.408} C_VEL
LIN {X 0,Y 367.55,Z 401.141,A -85,B 0,C 180,E1 17645.542,E2 17645.542} C_VEL
LIN {X 0,Y 366.984,Z 400.732,A -85,B 0,C 180,E1 17644.376,E2 17644.376} C_VEL
LIN {X 0,Y 366.73,Z 400.666,A -85,B 0,C 180,E1 17636.718,E2 17636.718} C_VEL
LIN {X 0,Y 367.527,Z 401.015,A -85,B 0,C 180,E1 17635.006,E2 17635.006} C_VEL
LIN {X 0,Y 368.804,Z 404.246,A -85,B 0,C 180,E1 17632.68,E2 17632.68} C_VEL
LIN {X 0,Y 372.366,Z 407.203,A -85,B 0,C 180,E1 17629.01,E2 17629.01} C_VEL
LIN {X 0,Y 373.448,Z 407.874,A -85,B 0,C 180,E1 17628.142,E2 17628.142} C_VEL
LIN {X 0,Y 375.524,Z 411.583,A -85,B 0,C 180,E1 17626.45,E2 17626.45} C_VEL
LIN {X 0,Y 379.055,Z 414.323,A -85,B 0,C 180,E1 17624.236,E2 17624.236} C_VEL
LIN {X 0,Y 381.623,Z 418.249,A -85,B 0,C 180,E1 17622.701,E2 17622.701} C_VEL
LIN {X 0,Y 384.385,Z 420.73,A -85,B 0,C 180,E1 17621.301,E2 17621.301} C_VEL
LIN {X 0,Y 387.527,Z 424.895,A -85,B 0,C 180,E1 17619.774,E2 17619.774} C_VEL
LIN {X 0,Y 389.61,Z 426.973,A -85,B 0,C 180,E1 17618.865,E2 17618.865} C_VEL
LIN {X 0,Y 393.24,Z 431.489,A -85,B 0,C 180,E1 17617.344,E2 17617.344} C_VEL
LIN {X 0,Y 400.505,Z 440.925,A -85,B 0,C 180,E1 17614.611,E2 17614.611} C_VEL
LIN {X 0,Y 410.502,Z 455.34,A -85,B 0,C 180,E1 17611.326,E2 17611.326} C_VEL
LIN {X 0,Y 420.82,Z 471.362,A -85,B 0,C 180,E1 17608.366,E2 17608.366} C_VEL
LIN {X 0,Y 427.146,Z 482.076,A -85,B 0,C 180,E1 17606.706,E2 17606.706} C_VEL
LIN {X 0,Y 416.635,Z 690.32,A -85,B 0,C 180,E1 17602.727,E2 17602.727} C_VEL
LIN {X 0,Y 414.061,Z 738.086,A -85,B 0,C 180,E1 17601.785,E2 17601.785} C_VEL
LIN {X 0,Y 411.558,Z 760.893,A -85,B 0,C 180,E1 17601.156,E2 17601.156} C_VEL
LIN {X 0,Y 408.41,Z 782.959,A -85,B 0,C 180,E1 17600.342,E2 17600.342} C_VEL
LIN {X 0,Y 404.662,Z 803.987,A -85,B 0,C 180,E1 17599.329,E2 17599.329} C_VEL
LIN {X 0,Y 400.087,Z 826.154,A -85,B 0,C 180,E1 17598,E2 17598} C_VEL
LIN {X 0,Y 395.387,Z 846.125,A -85,B 0,C 180,E1 17596.526,E2 17596.526} C_VEL
LIN {X 0,Y 389.892,Z 867.328,A -85,B 0,C 180,E1 17594.635,E2 17594.635} C_VEL
LIN {X 0,Y 384.719,Z 885.972,A -85,B 0,C 180,E1 17592.651,E2 17592.651} C_VEL
LIN {X 0,Y 379.279,Z 904.287,A -85,B 0,C 180,E1 17590.335,E2 17590.335} C_VEL
LIN {X 0,Y 374.21,Z 921.118,A -85,B 0,C 180,E1 17587.851,E2 17587.851} C_VEL
LIN {X 0,Y 369.261,Z 937.2,A -85,B 0,C 180,E1 17585.028,E2 17585.028} C_VEL
LIN {X 0,Y 364.742,Z 952.279,A -85,B 0,C 180,E1 17581.939,E2 17581.939} C_VEL
LIN {X 0,Y 361.22,Z 964.586,A -85,B 0,C 180,E1 17578.97,E2 17578.97} C_VEL
LIN {X 0,Y 357.826,Z 977.471,A -85,B 0,C 180,E1 17575.308,E2 17575.308} C_VEL
LIN {X 0,Y 355.477,Z 987.687,A -85,B 0,C 180,E1 17571.846,E2 17571.846} C_VEL
LIN {X 0,Y 353.794,Z 996.326,A -85,B 0,C 180,E1 17568.275,E2 17568.275} C_VEL
LIN {X 0,Y 352.764,Z 1003.278,A -85,B 0,C 180,E1 17564.778,E2 17564.778} C_VEL
LIN {X 0,Y 352.198,Z 1008.819,A -85,B 0,C 180,E1 17561.13,E2 17561.13} C_VEL
LIN {X 0,Y 351.987,Z 1012.532,A -85,B 0,C 180,E1 17557.836,E2 17557.836} C_VEL
LIN {X 0,Y 351.935,Z 1015.094,A -85,B 0,C 180,E1 17554.236,E2 17554.236} C_VEL
LIN {X 0,Y 351.93,Z 1016.06,A -85,B 0,C 180,E1 17551.14,E2 17551.14} C_VEL
LIN {X 0,Y 351.939,Z 1015.918,A -85,B 0,C 180,E1 17547.884,E2 17547.884} C_VEL
LIN {X 0,Y 351.937,Z 1014.217,A -85,B 0,C 180,E1 17544.294,E2 17544.294} C_VEL
LIN {X 0,Y 352.046,Z 1011.378,A -85,B 0,C 180,E1 17541.015,E2 17541.015} C_VEL
LIN {X 0,Y 352.411,Z 1006.498,A -85,B 0,C 180,E1 17537.217,E2 17537.217} C_VEL
LIN {X 0,Y 353.11,Z 1000.785,A -85,B 0,C 180,E1 17533.892,E2 17533.892} C_VEL
LIN {X 0,Y 354.504,Z 992.471,A -85,B 0,C 180,E1 17530.048,E2 17530.048} C_VEL
LIN {X 0,Y 356.369,Z 983.605,A -85,B 0,C 180,E1 17526.7,E2 17526.7} C_VEL
LIN {X 0,Y 359.091,Z 972.476,A -85,B 0,C 180,E1 17523.191,E2 17523.191} C_VEL
LIN {X 0,Y 362.316,Z 960.695,A -85,B 0,C 180,E1 17520.038,E2 17520.038} C_VEL
LIN {X 0,Y 366.313,Z 946.953,A -85,B 0,C 180,E1 17516.918,E2 17516.918} C_VEL
LIN {X 0,Y 370.931,Z 931.795,A -85,B 0,C 180,E1 17513.964,E2 17513.964} C_VEL
LIN {X 0,Y 375.996,Z 915.116,A -85,B 0,C 180,E1 17511.232,E2 17511.232} C_VEL
LIN {X 0,Y 381.337,Z 897.421,A -85,B 0,C 180,E1 17508.75,E2 17508.75} C_VEL
LIN {X 0,Y 386.494,Z 879.507,A -85,B 0,C 180,E1 17506.63,E2 17506.63} C_VEL
LIN {X 0,Y 392.165,Z 858.724,A -85,B 0,C 180,E1 17504.56,E2 17504.56} C_VEL
LIN {X 0,Y 396.72,Z 840.613,A -85,B 0,C 180,E1 17503.047,E2 17503.047} C_VEL
LIN {X 0,Y 401.542,Z 819.352,A -85,B 0,C 180,E1 17501.568,E2 17501.568} C_VEL
LIN {X 0,Y 405.392,Z 799.999,A -85,B 0,C 180,E1 17500.466,E2 17500.466} C_VEL
LIN {X 0,Y 409.322,Z 776.681,A -85,B 0,C 180,E1 17499.41,E2 17499.41} C_VEL
LIN {X 0,Y 412.041,Z 756.777,A -85,B 0,C 180,E1 17498.721,E2 17498.721} C_VEL
LIN {X 0,Y 414.439,Z 731.888,A -85,B 0,C 180,E1 17498.087,E2 17498.087} C_VEL
LIN {X 0,Y 424.386,Z 533.92,A -85,B 0,C 180,E1 17494.291,E2 17494.291} C_VEL
LIN {X 0,Y 426.996,Z 481.71,A -85,B 0,C 180,E1 17493.27,E2 17493.27} C_VEL
LIN {X 0,Y 417.725,Z 466.591,A -85,B 0,C 180,E1 17490.812,E2 17490.812} C_VEL
LIN {X 0,Y 409.17,Z 453.509,A -85,B 0,C 180,E1 17488.298,E2 17488.298} C_VEL
LIN {X 0,Y 401.811,Z 442.997,A -85,B 0,C 180,E1 17485.894,E2 17485.894} C_VEL
LIN {X 0,Y 396.993,Z 436.342,A -85,B 0,C 180,E1 17484.158,E2 17484.158} C_VEL
LIN {X 0,Y 393.13,Z 431.397,A -85,B 0,C 180,E1 17482.663,E2 17482.663} C_VEL
LIN {X 0,Y 389.497,Z 426.827,A -85,B 0,C 180,E1 17481.141,E2 17481.141} C_VEL
LIN {X 0,Y 384.947,Z 421.719,A -85,B 0,C 180,E1 17479.063,E2 17479.063} C_VEL
LIN {X 0,Y 383.911,Z 420.093,A -85,B 0,C 180,E1 17478.526,E2 17478.526} C_VEL
LIN {X 0,Y 380.575,Z 417.004,A -85,B 0,C 180,E1 17476.797,E2 17476.797} C_VEL
LIN {X 0,Y 378.669,Z 413.901,A -85,B 0,C 180,E1 17475.624,E2 17475.624} C_VEL
LIN {X 0,Y 375.266,Z 411.29,A -85,B 0,C 180,E1 17473.481,E2 17473.481} C_VEL
LIN {X 0,Y 373.154,Z 407.488,A -85,B 0,C 180,E1 17471.75,E2 17471.75} C_VEL
LIN {X 0,Y 369.616,Z 405.276,A -85,B 0,C 180,E1 17468.556,E2 17468.556} C_VEL
LIN {X 0,Y 367.621,Z 401.631,A -85,B 0,C 180,E1 17465.619,E2 17465.619} C_VEL
LIN {X 0,Y 367.333,Z 400.799,A -85,B 0,C 180,E1 17464.997,E2 17464.997} C_VEL
LIN {X 0,Y 366.166,Z 400.505,A -85,B 0,C 180,E1 17457.182,E2 17457.182} C_VEL
LIN {X 0,Y 367.521,Z 401.092,A -85,B 0,C 180,E1 17454.066,E2 17454.066} C_VEL
LIN {X 0,Y 369.02,Z 404.537,A -85,B 0,C 180,E1 17451.586,E2 17451.586} C_VEL
LIN {X 0,Y 372.256,Z 407.141,A -85,B 0,C 180,E1 17448.378,E2 17448.378} C_VEL
LIN {X 0,Y 373.398,Z 407.833,A -85,B 0,C 180,E1 17447.473,E2 17447.473} C_VEL
LIN {X 0,Y 375.242,Z 411.214,A -85,B 0,C 180,E1 17445.967,E2 17445.967} C_VEL
LIN {X 0,Y 378.998,Z 414.304,A -85,B 0,C 180,E1 17443.603,E2 17443.603} C_VEL
LIN {X 0,Y 381.589,Z 418.202,A -85,B 0,C 180,E1 17442.068,E2 17442.068} C_VEL
LIN {X 0,Y 384.442,Z 420.754,A -85,B 0,C 180,E1 17440.634,E2 17440.634} C_VEL
LIN {X 0,Y 387.523,Z 424.914,A -85,B 0,C 180,E1 17439.141,E2 17439.141} C_VEL
LIN {X 0,Y 389.533,Z 426.935,A -85,B 0,C 180,E1 17438.268,E2 17438.268} C_VEL
LIN {X 0,Y 393.09,Z 431.361,A -85,B 0,C 180,E1 17436.78,E2 17436.78} C_VEL
LIN {X 0,Y 399.176,Z 438.975,A -85,B 0,C 180,E1 17434.48,E2 17434.48} C_VEL
LIN {X 0,Y 403.883,Z 445.064,A -85,B 0,C 180,E1 17432.862,E2 17432.862} C_VEL
LIN {X 0,Y 410.756,Z 454.053,A -85,B 0,C 180,E1 17430.707,E2 17430.707} C_VEL
LIN {X 0,Y 420.671,Z 468.003,A -85,B 0,C 180,E1 17427.912,E2 17427.912} C_VEL
LIN {X 0,Y 426.996,Z 477.65,A -85,B 0,C 180,E1 17426.279,E2 17426.279} C_VEL
LIN {X 0,Y 416.404,Z 686.062,A -85,B 0,C 180,E1 17422.301,E2 17422.301} C_VEL
LIN {X 0,Y 414.376,Z 720.456,A -85,B 0,C 180,E1 17421.603,E2 17421.603} C_VEL
LIN {X 0,Y 412.048,Z 742.4,A -85,B 0,C 180,E1 17420.967,E2 17420.967} C_VEL
LIN {X 0,Y 408.7,Z 766.299,A -85,B 0,C 180,E1 17420.018,E2 17420.018} C_VEL
LIN {X 0,Y 405.253,Z 786.059,A -85,B 0,C 180,E1 17419.015,E2 17419.015} C_VEL
LIN {X 0,Y 400.823,Z 807.586,A -85,B 0,C 180,E1 17417.66,E2 17417.66} C_VEL
LIN {X 0,Y 396.48,Z 826.093,A -85,B 0,C 180,E1 17416.254,E2 17416.254} C_VEL
LIN {X 0,Y 391.059,Z 846.8,A -85,B 0,C 180,E1 17414.362,E2 17414.362} C_VEL
LIN {X 0,Y 385.968,Z 864.781,A -85,B 0,C 180,E1 17412.413,E2 17412.413} C_VEL
LIN {X 0,Y 380.603,Z 882.395,A -85,B 0,C 180,E1 17410.14,E2 17410.14} C_VEL
LIN {X 0,Y 375.34,Z 899.286,A -85,B 0,C 180,E1 17407.586,E2 17407.586} C_VEL
LIN {X 0,Y 370.407,Z 914.469,A -85,B 0,C 180,E1 17404.854,E2 17404.854} C_VEL
LIN {X 0,Y 365.619,Z 929.527,A -85,B 0,C 180,E1 17401.668,E2 17401.668} C_VEL
LIN {X 0,Y 361.973,Z 941.31,A -85,B 0,C 180,E1 17398.722,E2 17398.722} C_VEL
LIN {X 0,Y 358.573,Z 953.054,A -85,B 0,C 180,E1 17395.25,E2 17395.25} C_VEL
LIN {X 0,Y 356.13,Z 962.493,A -85,B 0,C 180,E1 17391.923,E2 17391.923} C_VEL
LIN {X 0,Y 354.931,Z 967.661,A -85,B 0,C 180,E1 17389.794,E2 17389.794} C_VEL
LIN {X 0,Y 353.419,Z 970.429,A -85,B 0,C 180,E1 17388.645,E2 17388.645} C_VEL
LIN {X 0,Y 346.04,Z 977.155,A -85,B 0,C 180,E1 17385.564,E2 17385.564} C_VEL
LIN {X 0,Y 345.011,Z 978.872,A -85,B 0,C 180,E1 17384.506,E2 17384.506} C_VEL
LIN {X 0,Y 344.366,Z 983.547,A -85,B 0,C 180,E1 17381.046,E2 17381.046} C_VEL
LIN {X 0,Y 344.041,Z 987.237,A -85,B 0,C 180,E1 17377.345,E2 17377.345} C_VEL
LIN {X 0,Y 343.954,Z 989.249,A -85,B 0,C 180,E1 17373.833,E2 17373.833} C_VEL
LIN {X 0,Y 343.929,Z 990.031,A -85,B 0,C 180,E1 17370.666,E2 17370.666} C_VEL
LIN {X 0,Y 343.937,Z 989.615,A -85,B 0,C 180,E1 17367,E2 17367} C_VEL
LIN {X 0,Y 344.012,Z 987.953,A -85,B 0,C 180,E1 17363.659,E2 17363.659} C_VEL
LIN {X 0,Y 344.237,Z 984.836,A -85,B 0,C 180,E1 17359.948,E2 17359.948} C_VEL
LIN {X 0,Y 344.822,Z 980.097,A -85,B 0,C 180,E1 17356.246,E2 17356.246} C_VEL
LIN {X 0,Y 345.919,Z 973.907,A -85,B 0,C 180,E1 17352.508,E2 17352.508} C_VEL
LIN {X 0,Y 347.597,Z 966.294,A -85,B 0,C 180,E1 17348.929,E2 17348.929} C_VEL
LIN {X 0,Y 350.181,Z 956.636,A -85,B 0,C 180,E1 17345.185,E2 17345.185} C_VEL
LIN {X 0,Y 353.344,Z 946.051,A -85,B 0,C 180,E1 17341.802,E2 17341.802} C_VEL
LIN {X 0,Y 357.568,Z 932.931,A -85,B 0,C 180,E1 17338.288,E2 17338.288} C_VEL
LIN {X 0,Y 361.987,Z 919.848,A -85,B 0,C 180,E1 17335.323,E2 17335.323} C_VEL
LIN {X 0,Y 367.121,Z 904.598,A -85,B 0,C 180,E1 17332.41,E2 17332.41} C_VEL
LIN {X 0,Y 372.521,Z 888.619,A -85,B 0,C 180,E1 17329.801,E2 17329.801} C_VEL
LIN {X 0,Y 378.103,Z 871.06,A -85,B 0,C 180,E1 17327.398,E2 17327.398} C_VEL
LIN {X 0,Y 383.858,Z 852.162,A -85,B 0,C 180,E1 17325.21,E2 17325.21} C_VEL
LIN {X 0,Y 388.958,Z 833.912,A -85,B 0,C 180,E1 17323.438,E2 17323.438} C_VEL
LIN {X 0,Y 394.381,Z 812.504,A -85,B 0,C 180,E1 17321.707,E2 17321.707} C_VEL
LIN {X 0,Y 398.39,Z 794.557,A -85,B 0,C 180,E1 17320.503,E2 17320.503} C_VEL
LIN {X 0,Y 402.653,Z 772.438,A -85,B 0,C 180,E1 17319.288,E2 17319.288} C_VEL
LIN {X 0,Y 405.737,Z 752.99,A -85,B 0,C 180,E1 17318.44,E2 17318.44} C_VEL
LIN {X 0,Y 408.636,Z 729.721,A -85,B 0,C 180,E1 17317.663,E2 17317.663} C_VEL
LIN {X 0,Y 410.443,Z 708.109,A -85,B 0,C 180,E1 17317.147,E2 17317.147} C_VEL
LIN {X 0,Y 421.435,Z 500.268,A -85,B 0,C 180,E1 17313.15,E2 17313.15} C_VEL
LIN {X 0,Y 422.41,Z 481.695,A -85,B 0,C 180,E1 17312.783,E2 17312.783} C_VEL
LIN {X 0,Y 412.982,Z 467.799,A -85,B 0,C 180,E1 17310.201,E2 17310.201} C_VEL
LIN {X 0,Y 405.719,Z 457.77,A -85,B 0,C 180,E1 17308,E2 17308} C_VEL
LIN {X 0,Y 398.972,Z 448.783,A -85,B 0,C 180,E1 17305.733,E2 17305.733} C_VEL
LIN {X 0,Y 395.028,Z 443.754,A -85,B 0,C 180,E1 17304.287,E2 17304.287} C_VEL
LIN {X 0,Y 391.058,Z 438.685,A -85,B 0,C 180,E1 17302.711,E2 17302.711} C_VEL
LIN {X 0,Y 387.362,Z 433.862,A -85,B 0,C 180,E1 17301.105,E2 17301.105} C_VEL
LIN {X 0,Y 383.573,Z 429.679,A -85,B 0,C 180,E1 17299.333,E2 17299.333} C_VEL
LIN {X 0,Y 382.2,Z 427.675,A -85,B 0,C 180,E1 17298.612,E2 17298.612} C_VEL
LIN {X 0,Y 378.839,Z 424.34,A -85,B 0,C 180,E1 17296.798,E2 17296.798} C_VEL
LIN {X 0,Y 377.097,Z 421.578,A -85,B 0,C 180,E1 17295.691,E2 17295.691} C_VEL
LIN {X 0,Y 373.529,Z 418.437,A -85,B 0,C 180,E1 17293.309,E2 17293.309} C_VEL
LIN {X 0,Y 371.967,Z 415.363,A -85,B 0,C 180,E1 17291.946,E2 17291.946} C_VEL
LIN {X 0,Y 368.421,Z 413.002,A -85,B 0,C 180,E1 17288.585,E2 17288.585} C_VEL
LIN {X 0,Y 366.578,Z 409.48,A -85,B 0,C 180,E1 17285.635,E2 17285.635} C_VEL
LIN {X 0,Y 366.316,Z 408.723,A -85,B 0,C 180,E1 17285.011,E2 17285.011} C_VEL
LIN {X 0,Y 365.643,Z 408.575,A -85,B 0,C 180,E1 17277.022,E2 17277.022} C_VEL
LIN {X 0,Y 366.46,Z 409.004,A -85,B 0,C 180,E1 17275.148,E2 17275.148} C_VEL
LIN {X 0,Y 368.052,Z 412.634,A -85,B 0,C 180,E1 17272.351,E2 17272.351} C_VEL
LIN {X 0,Y 371.785,Z 415.309,A -85,B 0,C 180,E1 17268.678,E2 17268.678} C_VEL
LIN {X 0,Y 374.657,Z 419.848,A -85,B 0,C 180,E1 17266.339,E2 17266.339} C_VEL
LIN {X 0,Y 377.582,Z 422.158,A -85,B 0,C 180,E1 17264.488,E2 17264.488} C_VEL
LIN {X 0,Y 380.389,Z 426.214,A -85,B 0,C 180,E1 17262.8,E2 17262.8} C_VEL
LIN {X 0,Y 382.693,Z 428.351,A -85,B 0,C 180,E1 17261.61,E2 17261.61} C_VEL
LIN {X 0,Y 385.945,Z 432.588,A -85,B 0,C 180,E1 17260.004,E2 17260.004} C_VEL
LIN {X 0,Y 387.829,Z 434.612,A -85,B 0,C 180,E1 17259.159,E2 17259.159} C_VEL
LIN {X 0,Y 391.592,Z 439.188,A -85,B 0,C 180,E1 17257.56,E2 17257.56} C_VEL
LIN {X 0,Y 398.566,Z 448.694,A -85,B 0,C 180,E1 17254.876,E2 17254.876} C_VEL
LIN {X 0,Y 407.634,Z 461.906,A -85,B 0,C 180,E1 17251.825,E2 17251.825} C_VEL
LIN {X 0,Y 417.769,Z 477.947,A -85,B 0,C 180,E1 17248.832,E2 17248.832} C_VEL
LIN {X 0,Y 422.533,Z 486.277,A -85,B 0,C 180,E1 17247.532,E2 17247.532} C_VEL
LIN {X 0,Y 411.437,Z 697.488,A -85,B 0,C 180,E1 17243.475,E2 17243.475} C_VEL
LIN {X 0,Y 409.081,Z 738.288,A -85,B 0,C 180,E1 17242.658,E2 17242.658} C_VEL
LIN {X 0,Y 406.526,Z 760.799,A -85,B 0,C 180,E1 17242.035,E2 17242.035} C_VEL
LIN {X 0,Y 403.159,Z 783.407,A -85,B 0,C 180,E1 17241.194,E2 17241.194} C_VEL
LIN {X 0,Y 399.414,Z 803.69,A -85,B 0,C 180,E1 17240.214,E2 17240.214} C_VEL
LIN {X 0,Y 394.721,Z 825.64,A -85,B 0,C 180,E1 17238.895,E2 17238.895} C_VEL
LIN {X 0,Y 389.97,Z 845.082,A -85,B 0,C 180,E1 17237.461,E2 17237.461} C_VEL
LIN {X 0,Y 384.051,Z 867.021,A -85,B 0,C 180,E1 17235.502,E2 17235.502} C_VEL
LIN {X 0,Y 378.563,Z 885.969,A -85,B 0,C 180,E1 17233.469,E2 17233.469} C_VEL
LIN {X 0,Y 373.127,Z 903.471,A -85,B 0,C 180,E1 17231.234,E2 17231.234} C_VEL
LIN {X 0,Y 367.739,Z 920.481,A -85,B 0,C 180,E1 17228.703,E2 17228.703} C_VEL
LIN {X 0,Y 362.691,Z 936.028,A -85,B 0,C 180,E1 17225.954,E2 17225.954} C_VEL
LIN {X 0,Y 358.113,Z 950.538,A -85,B 0,C 180,E1 17222.983,E2 17222.983} C_VEL
LIN {X 0,Y 354.096,Z 963.626,A -85,B 0,C 180,E1 17219.796,E2 17219.796} C_VEL
LIN {X 0,Y 350.57,Z 976.105,A -85,B 0,C 180,E1 17216.234,E2 17216.234} C_VEL
LIN {X 0,Y 348.04,Z 986.11,A -85,B 0,C 180,E1 17212.817,E2 17212.817} C_VEL
LIN {X 0,Y 346.034,Z 995.642,A -85,B 0,C 180,E1 17208.88,E2 17208.88} C_VEL
LIN {X 0,Y 344.929,Z 1002.348,A -85,B 0,C 180,E1 17205.466,E2 17205.466} C_VEL
LIN {X 0,Y 344.236,Z 1008.301,A -85,B 0,C 180,E1 17201.56,E2 17201.56} C_VEL
LIN {X 0,Y 344.017,Z 1012.065,A -85,B 0,C 180,E1 17198.187,E2 17198.187} C_VEL
LIN {X 0,Y 343.935,Z 1014.722,A -85,B 0,C 180,E1 17194.502,E2 17194.502} C_VEL
LIN {X 0,Y 343.941,Z 1015.737,A -85,B 0,C 180,E1 17191.333,E2 17191.333} C_VEL
LIN {X 0,Y 343.943,Z 1015.666,A -85,B 0,C 180,E1 17188.168,E2 17188.168} C_VEL
LIN {X 0,Y 343.939,Z 1014.151,A -85,B 0,C 180,E1 17184.496,E2 17184.496} C_VEL
LIN {X 0,Y 344.041,Z 1011.405,A -85,B 0,C 180,E1 17181.141,E2 17181.141} C_VEL
LIN {X 0,Y 344.379,Z 1006.977,A -85,B 0,C 180,E1 17177.425,E2 17177.425} C_VEL
LIN {X 0,Y 345.116,Z 1001.101,A -85,B 0,C 180,E1 17173.854,E2 17173.854} C_VEL
LIN {X 0,Y 346.479,Z 993.406,A -85,B 0,C 180,E1 17170.094,E2 17170.094} C_VEL
LIN {X 0,Y 348.489,Z 984.231,A -85,B 0,C 180,E1 17166.5,E2 17166.5} C_VEL
LIN {X 0,Y 351.478,Z 972.747,A -85,B 0,C 180,E1 17162.746,E2 17162.746} C_VEL
LIN {X 0,Y 354.861,Z 961.027,A -85,B 0,C 180,E1 17159.529,E2 17159.529} C_VEL
LIN {X 0,Y 359.307,Z 946.636,A -85,B 0,C 180,E1 17156.188,E2 17156.188} C_VEL
LIN {X 0,Y 364.104,Z 931.713,A -85,B 0,C 180,E1 17153.233,E2 17153.233} C_VEL
LIN {X 0,Y 369.388,Z 915.201,A -85,B 0,C 180,E1 17150.482,E2 17150.482} C_VEL
LIN {X 0,Y 374.929,Z 897.721,A -85,B 0,C 180,E1 17147.988,E2 17147.988} C_VEL
LIN {X 0,Y 380.317,Z 879.837,A -85,B 0,C 180,E1 17145.845,E2 17145.845} C_VEL
LIN {X 0,Y 386.211,Z 859.23,A -85,B 0,C 180,E1 17143.763,E2 17143.763} C_VEL
LIN {X 0,Y 390.932,Z 841.208,A -85,B 0,C 180,E1 17142.24,E2 17142.24} C_VEL
LIN {X 0,Y 396.173,Z 819.039,A -85,B 0,C 180,E1 17140.685,E2 17140.685} C_VEL
LIN {X 0,Y 400.182,Z 799.607,A -85,B 0,C 180,E1 17139.577,E2 17139.577} C_VEL
LIN {X 0,Y 404.27,Z 776.096,A -85,B 0,C 180,E1 17138.512,E2 17138.512} C_VEL
LIN {X 0,Y 407.15,Z 755.677,A -85,B 0,C 180,E1 17137.811,E2 17137.811} C_VEL
LIN {X 0,Y 409.545,Z 731.244,A -85,B 0,C 180,E1 17137.194,E2 17137.194} C_VEL
LIN {X 0,Y 419.972,Z 532.212,A -85,B 0,C 180,E1 17133.356,E2 17133.356} C_VEL
LIN {X 0,Y 422.448,Z 485.889,A -85,B 0,C 180,E1 17132.457,E2 17132.457} C_VEL
LIN {X 0,Y 413.428,Z 471.043,A -85,B 0,C 180,E1 17129.961,E2 17129.961} C_VEL
LIN {X 0,Y 404.621,Z 457.502,A -85,B 0,C 180,E1 17127.243,E2 17127.243} C_VEL
LIN {X 0,Y 396.543,Z 445.935,A -85,B 0,C 180,E1 17124.425,E2 17124.425} C_VEL
LIN {X 0,Y 391.132,Z 438.774,A -85,B 0,C 180,E1 17122.309,E2 17122.309} C_VEL
LIN {X 0,Y 387.412,Z 433.968,A -85,B 0,C 180,E1 17120.706,E2 17120.706} C_VEL
LIN {X 0,Y 383.238,Z 429.291,A -85,B 0,C 180,E1 17118.753,E2 17118.753} C_VEL
LIN {X 0,Y 382.077,Z 427.607,A -85,B 0,C 180,E1 17118.144,E2 17118.144} C_VEL
LIN {X 0,Y 378.714,Z 424.192,A -85,B 0,C 180,E1 17116.33,E2 17116.33} C_VEL
LIN {X 0,Y 377.208,Z 421.652,A -85,B 0,C 180,E1 17115.371,E2 17115.371} C_VEL
LIN {X 0,Y 373.776,Z 418.845,A -85,B 0,C 180,E1 17113.142,E2 17113.142} C_VEL
LIN {X 0,Y 371.801,Z 415.31,A -85,B 0,C 180,E1 17111.478,E2 17111.478} C_VEL
LIN {X 0,Y 368.243,Z 412.872,A -85,B 0,C 180,E1 17108.116,E2 17108.116} C_VEL
LIN {X 0,Y 366.418,Z 409.043,A -85,B 0,C 180,E1 17105.166,E2 17105.166} C_VEL
LIN {X 0,Y 365.724,Z 408.627,A -85,B 0,C 180,E1 17103.762,E2 17103.762} C_VEL
LIN {X 0,Y 365.382,Z 408.522,A -85,B 0,C 180,E1 17096.548,E2 17096.548} C_VEL
LIN {X 0,Y 366.42,Z 408.923,A -85,B 0,C 180,E1 17094.284,E2 17094.284} C_VEL
LIN {X 0,Y 367.923,Z 412.418,A -85,B 0,C 180,E1 17091.718,E2 17091.718} C_VEL
LIN {X 0,Y 371.112,Z 415.025,A -85,B 0,C 180,E1 17088.499,E2 17088.499} C_VEL
LIN {X 0,Y 372.083,Z 415.737,A -85,B 0,C 180,E1 17087.704,E2 17087.704} C_VEL
LIN {X 0,Y 374.165,Z 419.265,A -85,B 0,C 180,E1 17086.005,E2 17086.005} C_VEL
LIN {X 0,Y 377.524,Z 422.143,A -85,B 0,C 180,E1 17083.854,E2 17083.854} C_VEL
LIN {X 0,Y 380.356,Z 426.167,A -85,B 0,C 180,E1 17082.166,E2 17082.166} C_VEL
LIN {X 0,Y 382.747,Z 428.385,A -85,B 0,C 180,E1 17080.941,E2 17080.941} C_VEL
LIN {X 0,Y 386.098,Z 432.759,A -85,B 0,C 180,E1 17079.299,E2 17079.299} C_VEL
LIN {X 0,Y 387.752,Z 434.578,A -85,B 0,C 180,E1 17078.56,E2 17078.56} C_VEL
LIN {X 0,Y 391.62,Z 439.221,A -85,B 0,C 180,E1 17076.927,E2 17076.927} C_VEL
LIN {X 0,Y 395.821,Z 444.601,A -85,B 0,C 180,E1 17075.288,E2 17075.288} C_VEL
LIN {X 0,Y 402.214,Z 453.122,A -85,B 0,C 180,E1 17073.02,E2 17073.02} C_VEL
LIN {X 0,Y 410.748,Z 464.563,A -85,B 0,C 180,E1 17070.34,E2 17070.34} C_VEL
LIN {X 0,Y 420.699,Z 479.213,A -85,B 0,C 180,E1 17067.552,E2 17067.552} C_VEL
LIN {X 0,Y 422.382,Z 482.015,A -85,B 0,C 180,E1 17067.104,E2 17067.104} C_VEL
LIN {X 0,Y 411.383,Z 689.884,A -85,B 0,C 180,E1 17063.116,E2 17063.116} C_VEL
LIN {X 0,Y 409.342,Z 721.907,A -85,B 0,C 180,E1 17062.451,E2 17062.451} C_VEL
LIN {X 0,Y 406.956,Z 743.494,A -85,B 0,C 180,E1 17061.817,E2 17061.817} C_VEL
LIN {X 0,Y 403.582,Z 766.611,A -85,B 0,C 180,E1 17060.893,E2 17060.893} C_VEL
LIN {X 0,Y 399.891,Z 787.029,A -85,B 0,C 180,E1 17059.85,E2 17059.85} C_VEL
LIN {X 0,Y 395.253,Z 808.602,A -85,B 0,C 180,E1 17058.477,E2 17058.477} C_VEL
LIN {X 0,Y 390.692,Z 827.297,A -85,B 0,C 180,E1 17057.041,E2 17057.041} C_VEL
LIN {X 0,Y 385.277,Z 847.111,A -85,B 0,C 180,E1 17055.21,E2 17055.21} C_VEL
LIN {X 0,Y 380.06,Z 864.795,A -85,B 0,C 180,E1 17053.278,E2 17053.278} C_VEL
LIN {X 0,Y 374.387,Z 882.626,A -85,B 0,C 180,E1 17050.962,E2 17050.962} C_VEL
LIN {X 0,Y 369.03,Z 899.04,A -85,B 0,C 180,E1 17048.461,E2 17048.461} C_VEL
LIN {X 0,Y 363.734,Z 914.568,A -85,B 0,C 180,E1 17045.64,E2 17045.64} C_VEL
LIN {X 0,Y 358.837,Z 929.153,A -85,B 0,C 180,E1 17042.527,E2 17042.527} C_VEL
LIN {X 0,Y 354.856,Z 941.25,A -85,B 0,C 180,E1 17039.465,E2 17039.465} C_VEL
LIN {X 0,Y 351.123,Z 953.366,A -85,B 0,C 180,E1 17035.825,E2 17035.825} C_VEL
LIN {X 0,Y 348.503,Z 962.804,A -85,B 0,C 180,E1 17032.428,E2 17032.428} C_VEL
LIN {X 0,Y 346.433,Z 971.32,A -85,B 0,C 180,E1 17028.682,E2 17028.682} C_VEL
LIN {X 0,Y 345.16,Z 977.914,A -85,B 0,C 180,E1 17025.11,E2 17025.11} C_VEL
LIN {X 0,Y 345.011,Z 978.872,A -85,B 0,C 180,E1 17024.506,E2 17024.506} C_VEL
LIN {X 0,Y 343.754,Z 980.77,A -85,B 0,C 180,E1 17023.27,E2 17023.27} C_VEL
LIN {X 0,Y 339.128,Z 983.901,A -85,B 0,C 180,E1 17021.114,E2 17021.114} C_VEL
LIN {X 0,Y 336.497,Z 985.769,A -85,B 0,C 180,E1 17019.495,E2 17019.495} C_VEL
LIN {X 0,Y 336.169,Z 986.37,A -85,B 0,C 180,E1 17018.841,E2 17018.841} C_VEL
LIN {X 0,Y 335.989,Z 989.074,A -85,B 0,C 180,E1 17015.121,E2 17015.121} C_VEL
LIN {X 0,Y 335.951,Z 990.22,A -85,B 0,C 180,E1 17011.534,E2 17011.534} C_VEL
LIN {X 0,Y 335.954,Z 990.21,A -85,B 0,C 180,E1 17008.294,E2 17008.294} C_VEL
LIN {X 0,Y 335.997,Z 988.803,A -85,B 0,C 180,E1 17004.365,E2 17004.365} C_VEL
LIN {X 0,Y 336.177,Z 986.229,A -85,B 0,C 180,E1 17000.909,E2 17000.909} C_VEL
LIN {X 0,Y 336.666,Z 982.128,A -85,B 0,C 180,E1 16997.131,E2 16997.131} C_VEL
LIN {X 0,Y 337.664,Z 976.314,A -85,B 0,C 180,E1 16993.309,E2 16993.309} C_VEL
LIN {X 0,Y 339.436,Z 968.574,A -85,B 0,C 180,E1 16989.302,E2 16989.302} C_VEL
LIN {X 0,Y 341.717,Z 960.208,A -85,B 0,C 180,E1 16985.82,E2 16985.82} C_VEL
LIN {X 0,Y 345.145,Z 949.163,A -85,B 0,C 180,E1 16982.014,E2 16982.014} C_VEL
LIN {X 0,Y 348.955,Z 937.888,A -85,B 0,C 180,E1 16978.764,E2 16978.764} C_VEL
LIN {X 0,Y 353.575,Z 924.695,A -85,B 0,C 180,E1 16975.562,E2 16975.562} C_VEL
LIN {X 0,Y 358.736,Z 910.296,A -85,B 0,C 180,E1 16972.588,E2 16972.588} C_VEL
LIN {X 0,Y 364.3,Z 894.433,A -85,B 0,C 180,E1 16969.841,E2 16969.841} C_VEL
LIN {X 0,Y 370.187,Z 877.368,A -85,B 0,C 180,E1 16967.323,E2 16967.323} C_VEL
LIN {X 0,Y 375.783,Z 859.944,A -85,B 0,C 180,E1 16965.169,E2 16965.169} C_VEL
LIN {X 0,Y 381.612,Z 840.636,A -85,B 0,C 180,E1 16963.145,E2 16963.145} C_VEL
LIN {X 0,Y 386.881,Z 821.284,A -85,B 0,C 180,E1 16961.462,E2 16961.462} C_VEL
LIN {X 0,Y 392.195,Z 799.341,A -85,B 0,C 180,E1 16959.889,E2 16959.889} C_VEL
LIN {X 0,Y 396.464,Z 778.893,A -85,B 0,C 180,E1 16958.698,E2 16958.698} C_VEL
LIN {X 0,Y 400.279,Z 756.658,A -85,B 0,C 180,E1 16957.675,E2 16957.675} C_VEL
LIN {X 0,Y 403.25,Z 734.982,A -85,B 0,C 180,E1 16956.904,E2 16956.904} C_VEL
LIN {X 0,Y 405.414,Z 711.855,A -85,B 0,C 180,E1 16956.319,E2 16956.319} C_VEL
LIN {X 0,Y 416.643,Z 508.733,A -85,B 0,C 180,E1 16952.387,E2 16952.387} C_VEL
LIN {X 0,Y 417.841,Z 486.027,A -85,B 0,C 180,E1 16951.927,E2 16951.927} C_VEL
LIN {X 0,Y 408.668,Z 472.345,A -85,B 0,C 180,E1 16949.297,E2 16949.297} C_VEL
LIN {X 0,Y 400.669,Z 461.23,A -85,B 0,C 180,E1 16946.732,E2 16946.732} C_VEL
LIN {X 0,Y 393.712,Z 451.879,A -85,B 0,C 180,E1 16944.214,E2 16944.214} C_VEL
LIN {X 0,Y 388.748,Z 445.712,A -85,B 0,C 180,E1 16942.215,E2 16942.215} C_VEL
LIN {X 0,Y 384.823,Z 440.697,A -85,B 0,C 180,E1 16940.455,E2 16940.455} C_VEL
LIN {X 0,Y 381.278,Z 436.283,A -85,B 0,C 180,E1 16938.699,E2 16938.699} C_VEL
LIN {X 0,Y 380.109,Z 434.953,A -85,B 0,C 180,E1 16938.083,E2 16938.083} C_VEL
LIN {X 0,Y 376.777,Z 431.161,A -85,B 0,C 180,E1 16936.179,E2 16936.179} C_VEL
LIN {X 0,Y 375.652,Z 429.321,A -85,B 0,C 180,E1 16935.437,E2 16935.437} C_VEL
LIN {X 0,Y 372.162,Z 426.127,A -85,B 0,C 180,E1 16933.043,E2 16933.043} C_VEL
LIN {X 0,Y 370.626,Z 423.183,A -85,B 0,C 180,E1 16931.674,E2 16931.674} C_VEL
LIN {X 0,Y 367.196,Z 420.743,A -85,B 0,C 180,E1 16928.298,E2 16928.298} C_VEL
LIN {X 0,Y 365.426,Z 417.047,A -85,B 0,C 180,E1 16925.26,E2 16925.26} C_VEL
LIN {X 0,Y 365.111,Z 416.627,A -85,B 0,C 180,E1 16924.555,E2 16924.555} C_VEL
LIN {X 0,Y 364.725,Z 416.532,A -85,B 0,C 180,E1 16916.857,E2 16916.857} C_VEL
LIN {X 0,Y 365.398,Z 416.969,A -85,B 0,C 180,E1 16915.292,E2 16915.292} C_VEL
LIN {X 0,Y 367.321,Z 420.952,A -85,B 0,C 180,E1 16912.021,E2 16912.021} C_VEL
LIN {X 0,Y 370.8,Z 423.491,A -85,B 0,C 180,E1 16908.648,E2 16908.648} C_VEL
LIN {X 0,Y 373.055,Z 427.315,A -85,B 0,C 180,E1 16906.753,E2 16906.753} C_VEL
LIN {X 0,Y 376.065,Z 429.854,A -85,B 0,C 180,E1 16904.779,E2 16904.779} C_VEL
LIN {X 0,Y 379.024,Z 434.034,A -85,B 0,C 180,E1 16902.974,E2 16902.974} C_VEL
LIN {X 0,Y 381.014,Z 435.954,A -85,B 0,C 180,E1 16901.922,E2 16901.922} C_VEL
LIN {X 0,Y 384.523,Z 440.425,A -85,B 0,C 180,E1 16900.164,E2 16900.164} C_VEL
LIN {X 0,Y 386.06,Z 442.231,A -85,B 0,C 180,E1 16899.456,E2 16899.456} C_VEL
LIN {X 0,Y 390.671,Z 448.157,A -85,B 0,C 180,E1 16897.465,E2 16897.465} C_VEL
LIN {X 0,Y 396.191,Z 455.714,A -85,B 0,C 180,E1 16895.313,E2 16895.313} C_VEL
LIN {X 0,Y 405.195,Z 469.129,A -85,B 0,C 180,E1 16892.201,E2 16892.201} C_VEL
LIN {X 0,Y 414.746,Z 484.531,A -85,B 0,C 180,E1 16889.305,E2 16889.305} C_VEL
LIN {X 0,Y 418.012,Z 490.438,A -85,B 0,C 180,E1 16888.377,E2 16888.377} C_VEL
LIN {X 0,Y 406.374,Z 703.413,A -85,B 0,C 180,E1 16884.267,E2 16884.267} C_VEL
LIN {X 0,Y 404.159,Z 738.863,A -85,B 0,C 180,E1 16883.543,E2 16883.543} C_VEL
LIN {X 0,Y 401.564,Z 760.913,A -85,B 0,C 180,E1 16882.928,E2 16882.928} C_VEL
LIN {X 0,Y 397.999,Z 783.855,A -85,B 0,C 180,E1 16882.069,E2 16882.069} C_VEL
LIN {X 0,Y 394.266,Z 803.392,A -85,B 0,C 180,E1 16881.121,E2 16881.121} C_VEL
LIN {X 0,Y 389.404,Z 825.339,A -85,B 0,C 180,E1 16879.8,E2 16879.8} C_VEL
LIN {X 0,Y 384.516,Z 844.612,A -85,B 0,C 180,E1 16878.375,E2 16878.375} C_VEL
LIN {X 0,Y 378.529,Z 865.974,A -85,B 0,C 180,E1 16876.469,E2 16876.469} C_VEL
LIN {X 0,Y 373.033,Z 884.128,A -85,B 0,C 180,E1 16874.523,E2 16874.523} C_VEL
LIN {X 0,Y 367.189,Z 902.293,A -85,B 0,C 180,E1 16872.213,E2 16872.213} C_VEL
LIN {X 0,Y 361.818,Z 918.439,A -85,B 0,C 180,E1 16869.805,E2 16869.805} C_VEL
LIN {X 0,Y 356.223,Z 934.856,A -85,B 0,C 180,E1 16866.913,E2 16866.913} C_VEL
LIN {X 0,Y 351.36,Z 949.475,A -85,B 0,C 180,E1 16863.897,E2 16863.897} C_VEL
LIN {X 0,Y 347.033,Z 962.664,A -85,B 0,C 180,E1 16860.658,E2 16860.658} C_VEL
LIN {X 0,Y 343.398,Z 974.738,A -85,B 0,C 180,E1 16857.199,E2 16857.199} C_VEL
LIN {X 0,Y 340.494,Z 985.329,A -85,B 0,C 180,E1 16853.536,E2 16853.536} C_VEL
LIN {X 0,Y 338.291,Z 994.97,A -85,B 0,C 180,E1 16849.509,E2 16849.509} C_VEL
LIN {X 0,Y 337.074,Z 1001.729,A -85,B 0,C 180,E1 16846.012,E2 16846.012} C_VEL
LIN {X 0,Y 336.285,Z 1007.81,A -85,B 0,C 180,E1 16841.989,E2 16841.989} C_VEL
LIN {X 0,Y 336.031,Z 1011.597,A -85,B 0,C 180,E1 16838.555,E2 16838.555} C_VEL
LIN {X 0,Y 335.937,Z 1014.35,A -85,B 0,C 180,E1 16834.78,E2 16834.78} C_VEL
LIN {X 0,Y 335.947,Z 1015.437,A -85,B 0,C 180,E1 16831.365,E2 16831.365} C_VEL
LIN {X 0,Y 335.949,Z 1015.366,A -85,B 0,C 180,E1 16828.125,E2 16828.125} C_VEL
LIN {X 0,Y 335.942,Z 1013.849,A -85,B 0,C 180,E1 16824.365,E2 16824.365} C_VEL
LIN {X 0,Y 336.051,Z 1011.101,A -85,B 0,C 180,E1 16820.929,E2 16820.929} C_VEL
LIN {X 0,Y 336.423,Z 1006.657,A -85,B 0,C 180,E1 16817.114,E2 16817.114} C_VEL
LIN {X 0,Y 337.223,Z 1000.792,A -85,B 0,C 180,E1 16813.465,E2 16813.465} C_VEL
LIN {X 0,Y 338.693,Z 993.094,A -85,B 0,C 180,E1 16809.617,E2 16809.617} C_VEL
LIN {X 0,Y 340.855,Z 983.917,A -85,B 0,C 180,E1 16805.94,E2 16805.94} C_VEL
LIN {X 0,Y 344.11,Z 972.217,A -85,B 0,C 180,E1 16802.043,E2 16802.043} C_VEL
LIN {X 0,Y 347.866,Z 960.062,A -85,B 0,C 180,E1 16798.656,E2 16798.656} C_VEL
LIN {X 0,Y 352.472,Z 945.958,A -85,B 0,C 180,E1 16795.349,E2 16795.349} C_VEL
LIN {X 0,Y 357.736,Z 930.512,A -85,B 0,C 180,E1 16792.264,E2 16792.264} C_VEL
LIN {X 0,Y 363.28,Z 913.969,A -85,B 0,C 180,E1 16789.499,E2 16789.499} C_VEL
LIN {X 0,Y 369.358,Z 895.557,A -85,B 0,C 180,E1 16786.887,E2 16786.887} C_VEL
LIN {X 0,Y 375.097,Z 877.398,A -85,B 0,C 180,E1 16784.725,E2 16784.725} C_VEL
LIN {X 0,Y 381.01,Z 857.278,A -85,B 0,C 180,E1 16782.719,E2 16782.719} C_VEL
LIN {X 0,Y 386.233,Z 838.036,A -85,B 0,C 180,E1 16781.112,E2 16781.112} C_VEL
LIN {X 0,Y 391.335,Z 816.719,A -85,B 0,C 180,E1 16779.652,E2 16779.652} C_VEL
LIN {X 0,Y 395.83,Z 795.5,A -85,B 0,C 180,E1 16778.468,E2 16778.468} C_VEL
LIN {X 0,Y 399.744,Z 772.764,A -85,B 0,C 180,E1 16777.486,E2 16777.486} C_VEL
LIN {X 0,Y 402.983,Z 749.448,A -85,B 0,C 180,E1 16776.731,E2 16776.731} C_VEL
LIN {X 0,Y 405.016,Z 726.841,A -85,B 0,C 180,E1 16776.199,E2 16776.199} C_VEL
LIN {X 0,Y 416.109,Z 522.776,A -85,B 0,C 180,E1 16772.252,E2 16772.252} C_VEL
LIN {X 0,Y 417.877,Z 490.009,A -85,B 0,C 180,E1 16771.601,E2 16771.601} C_VEL
LIN {X 0,Y 409.949,Z 476.769,A -85,B 0,C 180,E1 16769.315,E2 16769.315} C_VEL
LIN {X 0,Y 401.827,Z 464.108,A -85,B 0,C 180,E1 16766.724,E2 16766.724} C_VEL
LIN {X 0,Y 394.115,Z 452.825,A -85,B 0,C 180,E1 16763.948,E2 16763.948} C_VEL
LIN {X 0,Y 388.98,Z 445.975,A -85,B 0,C 180,E1 16761.883,E2 16761.883} C_VEL
LIN {X 0,Y 384.71,Z 440.606,A -85,B 0,C 180,E1 16759.984,E2 16759.984} C_VEL
LIN {X 0,Y 381.085,Z 436.114,A -85,B 0,C 180,E1 16758.193,E2 16758.193} C_VEL
LIN {X 0,Y 379.701,Z 434.657,A -85,B 0,C 180,E1 16757.469,E2 16757.469} C_VEL
LIN {X 0,Y 376.534,Z 430.797,A -85,B 0,C 180,E1 16755.636,E2 16755.636} C_VEL
LIN {X 0,Y 375.508,Z 429.25,A -85,B 0,C 180,E1 16754.968,E2 16754.968} C_VEL
LIN {X 0,Y 372.299,Z 426.398,A -85,B 0,C 180,E1 16752.801,E2 16752.801} C_VEL
LIN {X 0,Y 370.457,Z 423.124,A -85,B 0,C 180,E1 16751.205,E2 16751.205} C_VEL
LIN {X 0,Y 366.895,Z 420.449,A -85,B 0,C 180,E1 16747.673,E2 16747.673} C_VEL
LIN {X 0,Y 365.214,Z 416.656,A -85,B 0,C 180,E1 16744.711,E2 16744.711} C_VEL
LIN {X 0,Y 364.263,Z 416.403,A -85,B 0,C 180,E1 16737.01,E2 16737.01} C_VEL
LIN {X 0,Y 365.354,Z 416.878,A -85,B 0,C 180,E1 16734.424,E2 16734.424} C_VEL
LIN {X 0,Y 366.827,Z 420.3,A -85,B 0,C 180,E1 16731.851,E2 16731.851} C_VEL
LIN {X 0,Y 370.153,Z 422.995,A -85,B 0,C 180,E1 16728.469,E2 16728.469} C_VEL
LIN {X 0,Y 370.779,Z 423.599,A -85,B 0,C 180,E1 16727.937,E2 16727.937} C_VEL
LIN {X 0,Y 372.985,Z 427.185,A -85,B 0,C 180,E1 16726.118,E2 16726.118} C_VEL
LIN {X 0,Y 376.006,Z 429.841,A -85,B 0,C 180,E1 16724.143,E2 16724.143} C_VEL
LIN {X 0,Y 378.991,Z 433.988,A -85,B 0,C 180,E1 16722.338,E2 16722.338} C_VEL
LIN {X 0,Y 381.065,Z 435.996,A -85,B 0,C 180,E1 16721.251,E2 16721.251} C_VEL
LIN {X 0,Y 384.52,Z 440.453,A -85,B 0,C 180,E1 16719.528,E2 16719.528} C_VEL
LIN {X 0,Y 386.06,Z 442.318,A -85,B 0,C 180,E1 16718.82,E2 16718.82} C_VEL
LIN {X 0,Y 390.531,Z 448.006,A -85,B 0,C 180,E1 16716.898,E2 16716.898} C_VEL
LIN {X 0,Y 395.184,Z 454.039,A -85,B 0,C 180,E1 16715.085,E2 16715.085} C_VEL
LIN {X 0,Y 401.635,Z 462.539,A -85,B 0,C 180,E1 16712.818,E2 16712.818} C_VEL
LIN {X 0,Y 410.911,Z 475.611,A -85,B 0,C 180,E1 16709.917,E2 16709.917} C_VEL
LIN {X 0,Y 417.868,Z 486.214,A -85,B 0,C 180,E1 16707.95,E2 16707.95} C_VEL
LIN {X 0,Y 406.423,Z 694.2,A -85,B 0,C 180,E1 16703.94,E2 16703.94} C_VEL
LIN {X 0,Y 404.302,Z 724.328,A -85,B 0,C 180,E1 16703.294,E2 16703.294} C_VEL
LIN {X 0,Y 401.776,Z 746.118,A -85,B 0,C 180,E1 16702.635,E2 16702.635} C_VEL
LIN {X 0,Y 398.305,Z 768.394,A -85,B 0,C 180,E1 16701.72,E2 16701.72} C_VEL
LIN {X 0,Y 394.384,Z 789.233,A -85,B 0,C 180,E1 16700.638,E2 16700.638} C_VEL
LIN {X 0,Y 389.697,Z 809.908,A -85,B 0,C 180,E1 16699.295,E2 16699.295} C_VEL
LIN {X 0,Y 384.527,Z 830.255,A -85,B 0,C 180,E1 16697.703,E2 16697.703} C_VEL
LIN {X 0,Y 378.925,Z 849.602,A -85,B 0,C 180,E1 16695.859,E2 16695.859} C_VEL
LIN {X 0,Y 372.964,Z 868.719,A -85,B 0,C 180,E1 16693.697,E2 16693.697} C_VEL
LIN {X 0,Y 367.303,Z 885.675,A -85,B 0,C 180,E1 16691.407,E2 16691.407} C_VEL
LIN {X 0,Y 361.411,Z 902.645,A -85,B 0,C 180,E1 16688.694,E2 16688.694} C_VEL
LIN {X 0,Y 356.183,Z 917.373,A -85,B 0,C 180,E1 16685.917,E2 16685.917} C_VEL
LIN {X 0,Y 351.145,Z 931.527,A -85,B 0,C 180,E1 16682.748,E2 16682.748} C_VEL
LIN {X 0,Y 346.751,Z 944.401,A -85,B 0,C 180,E1 16679.349,E2 16679.349} C_VEL
LIN {X 0,Y 343.064,Z 955.689,A -85,B 0,C 180,E1 16675.734,E2 16675.734} C_VEL
LIN {X 0,Y 340.054,Z 966.097,A -85,B 0,C 180,E1 16671.699,E2 16671.699} C_VEL
LIN {X 0,Y 338.209,Z 973.69,A -85,B 0,C 180,E1 16668.082,E2 16668.082} C_VEL
LIN {X 0,Y 336.938,Z 980.272,A -85,B 0,C 180,E1 16664.081,E2 16664.081} C_VEL
LIN {X 0,Y 336.297,Z 984.852,A -85,B 0,C 180,E1 16660.447,E2 16660.447} C_VEL
LIN {X 0,Y 336.169,Z 986.37,A -85,B 0,C 180,E1 16658.841,E2 16658.841} C_VEL
LIN {X 0,Y 335.083,Z 987.576,A -85,B 0,C 180,E1 16657.543,E2 16657.543} C_VEL
LIN {X 0,Y 328.584,Z 989.86,A -85,B 0,C 180,E1 16653.957,E2 16653.957} C_VEL
LIN {X 0,Y 327.951,Z 990.275,A -85,B 0,C 180,E1 16652.892,E2 16652.892} C_VEL
LIN {X 0,Y 327.939,Z 990.62,A -85,B 0,C 180,E1 16649.126,E2 16649.126} C_VEL
LIN {X 0,Y 327.974,Z 989.82,A -85,B 0,C 180,E1 16645.804,E2 16645.804} C_VEL
LIN {X 0,Y 328.11,Z 987.633,A -85,B 0,C 180,E1 16641.942,E2 16641.942} C_VEL
LIN {X 0,Y 328.483,Z 984.06,A -85,B 0,C 180,E1 16638.233,E2 16638.233} C_VEL
LIN {X 0,Y 329.356,Z 978.971,A -85,B 0,C 180,E1 16634.326,E2 16634.326} C_VEL
LIN {X 0,Y 330.889,Z 972.114,A -85,B 0,C 180,E1 16630.404,E2 16630.404} C_VEL
LIN {X 0,Y 333.254,Z 963.649,A -85,B 0,C 180,E1 16626.484,E2 16626.484} C_VEL
LIN {X 0,Y 336.241,Z 954.234,A -85,B 0,C 180,E1 16622.94,E2 16622.94} C_VEL
LIN {X 0,Y 340.54,Z 941.927,A -85,B 0,C 180,E1 16619.085,E2 16619.085} C_VEL
LIN {X 0,Y 345.143,Z 929.425,A -85,B 0,C 180,E1 16615.809,E2 16615.809} C_VEL
LIN {X 0,Y 350.317,Z 915.59,A -85,B 0,C 180,E1 16612.77,E2 16612.77} C_VEL
LIN {X 0,Y 355.914,Z 900.652,A -85,B 0,C 180,E1 16609.965,E2 16609.965} C_VEL
LIN {X 0,Y 361.802,Z 884.307,A -85,B 0,C 180,E1 16607.39,E2 16607.39} C_VEL
LIN {X 0,Y 367.91,Z 866.84,A -85,B 0,C 180,E1 16605.047,E2 16605.047} C_VEL
LIN {X 0,Y 373.72,Z 848.684,A -85,B 0,C 180,E1 16603.019,E2 16603.019} C_VEL
LIN {X 0,Y 379.415,Z 829.604,A -85,B 0,C 180,E1 16601.21,E2 16601.21} C_VEL
LIN {X 0,Y 384.538,Z 810.107,A -85,B 0,C 180,E1 16599.685,E2 16599.685} C_VEL
LIN {X 0,Y 389.399,Z 789.395,A -85,B 0,C 180,E1 16598.34,E2 16598.34} C_VEL
LIN {X 0,Y 393.475,Z 768.45,A -85,B 0,C 180,E1 16597.252,E2 16597.252} C_VEL
LIN {X 0,Y 397.095,Z 745.797,A -85,B 0,C 180,E1 16596.327,E2 16596.327} C_VEL
LIN {X 0,Y 399.697,Z 723.976,A -85,B 0,C 180,E1 16595.672,E2 16595.672} C_VEL
LIN {X 0,Y 401.908,Z 693.081,A -85,B 0,C 180,E1 16595.014,E2 16595.014} C_VEL
LIN {X 0,Y 413.507,Z 490.491,A -85,B 0,C 180,E1 16591.089,E2 16591.089} C_VEL
LIN {X 0,Y 404.175,Z 476.605,A -85,B 0,C 180,E1 16588.287,E2 16588.287} C_VEL
LIN {X 0,Y 395.348,Z 464.162,A -85,B 0,C 180,E1 16585.264,E2 16585.264} C_VEL
LIN {X 0,Y 390.182,Z 457.557,A -85,B 0,C 180,E1 16583.283,E2 16583.283} C_VEL
LIN {X 0,Y 386.796,Z 453.081,A -85,B 0,C 180,E1 16581.854,E2 16581.854} C_VEL
LIN {X 0,Y 382.942,Z 448.104,A -85,B 0,C 180,E1 16580.081,E2 16580.081} C_VEL
LIN {X 0,Y 379.351,Z 443.428,A -85,B 0,C 180,E1 16578.24,E2 16578.24} C_VEL
LIN {X 0,Y 375.319,Z 438.896,A -85,B 0,C 180,E1 16575.926,E2 16575.926} C_VEL
LIN {X 0,Y 374.216,Z 437.056,A -85,B 0,C 180,E1 16575.18,E2 16575.18} C_VEL
LIN {X 0,Y 370.711,Z 433.68,A -85,B 0,C 180,E1 16572.699,E2 16572.699} C_VEL
LIN {X 0,Y 369.294,Z 430.994,A -85,B 0,C 180,E1 16571.4,E2 16571.4} C_VEL
LIN {X 0,Y 365.864,Z 428.337,A -85,B 0,C 180,E1 16567.854,E2 16567.854} C_VEL
LIN {X 0,Y 364.215,Z 424.58,A -85,B 0,C 180,E1 16564.724,E2 16564.724} C_VEL
LIN {X 0,Y 363.751,Z 424.473,A -85,B 0,C 180,E1 16556.849,E2 16556.849} C_VEL
LIN {X 0,Y 364.34,Z 424.916,A -85,B 0,C 180,E1 16555.436,E2 16555.436} C_VEL
LIN {X 0,Y 366.346,Z 428.964,A -85,B 0,C 180,E1 16551.999,E2 16551.999} C_VEL
LIN {X 0,Y 369.546,Z 431.416,A -85,B 0,C 180,E1 16548.846,E2 16548.846} C_VEL
LIN {X 0,Y 371.876,Z 435.232,A -85,B 0,C 180,E1 16546.868,E2 16546.868} C_VEL
LIN {X 0,Y 374.608,Z 437.628,A -85,B 0,C 180,E1 16545.039,E2 16545.039} C_VEL
LIN {X 0,Y 377.662,Z 441.851,A -85,B 0,C 180,E1 16543.148,E2 16543.148} C_VEL
LIN {X 0,Y 379.412,Z 443.657,A -85,B 0,C 180,E1 16542.201,E2 16542.201} C_VEL
LIN {X 0,Y 383.105,Z 448.259,A -85,B 0,C 180,E1 16540.326,E2 16540.326} C_VEL
LIN {X 0,Y 388.599,Z 455.419,A -85,B 0,C 180,E1 16537.856,E2 16537.856} C_VEL
LIN {X 0,Y 394.014,Z 463.02,A -85,B 0,C 180,E1 16535.687,E2 16535.687} C_VEL
LIN {X 0,Y 402.481,Z 475.858,A -85,B 0,C 180,E1 16532.68,E2 16532.68} C_VEL
LIN {X 0,Y 411.753,Z 491.113,A -85,B 0,C 180,E1 16529.784,E2 16529.784} C_VEL
LIN {X 0,Y 413.585,Z 494.567,A -85,B 0,C 180,E1 16529.241,E2 16529.241} C_VEL
LIN {X 0,Y 401.443,Z 708.366,A -85,B 0,C 180,E1 16525.097,E2 16525.097} C_VEL
LIN {X 0,Y 399.24,Z 740.319,A -85,B 0,C 180,E1 16524.427,E2 16524.427} C_VEL
LIN {X 0,Y 396.61,Z 761.704,A -85,B 0,C 180,E1 16523.823,E2 16523.823} C_VEL
LIN {X 0,Y 392.914,Z 784.411,A -85,B 0,C 180,E1 16522.962,E2 16522.962} C_VEL
LIN {X 0,Y 389.216,Z 803.095,A -85,B 0,C 180,E1 16522.052,E2 16522.052} C_VEL
LIN {X 0,Y 384.187,Z 825.039,A -85,B 0,C 180,E1 16520.73,E2 16520.73} C_VEL
LIN {X 0,Y 379.12,Z 844.309,A -85,B 0,C 180,E1 16519.301,E2 16519.301} C_VEL
LIN {X 0,Y 372.896,Z 865.669,A -85,B 0,C 180,E1 16517.387,E2 16517.387} C_VEL
LIN {X 0,Y 367.108,Z 884.003,A -85,B 0,C 180,E1 16515.41,E2 16515.41} C_VEL
LIN {X 0,Y 360.756,Z 902.852,A -85,B 0,C 180,E1 16512.979,E2 16512.979} C_VEL
LIN {X 0,Y 354.85,Z 919.86,A -85,B 0,C 180,E1 16510.391,E2 16510.391} C_VEL
LIN {X 0,Y 349.132,Z 935.725,A -85,B 0,C 180,E1 16507.507,E2 16507.507} C_VEL
LIN {X 0,Y 343.897,Z 950.626,A -85,B 0,C 180,E1 16504.332,E2 16504.332} C_VEL
LIN {X 0,Y 339.411,Z 963.647,A -85,B 0,C 180,E1 16501.029,E2 16501.029} C_VEL
LIN {X 0,Y 335.299,Z 976.533,A -85,B 0,C 180,E1 16497.142,E2 16497.142} C_VEL
LIN {X 0,Y 332.417,Z 986.74,A -85,B 0,C 180,E1 16493.454,E2 16493.454} C_VEL
LIN {X 0,Y 330.334,Z 995.387,A -85,B 0,C 180,E1 16489.63,E2 16489.63} C_VEL
LIN {X 0,Y 328.98,Z 1002.668,A -85,B 0,C 180,E1 16485.692,E2 16485.692} C_VEL
LIN {X 0,Y 328.279,Z 1007.905,A -85,B 0,C 180,E1 16481.952,E2 16481.952} C_VEL
LIN {X 0,Y 328.026,Z 1011.625,A -85,B 0,C 180,E1 16478.413,E2 16478.413} C_VEL
LIN {X 0,Y 327.942,Z 1014.192,A -85,B 0,C 180,E1 16474.547,E2 16474.547} C_VEL
LIN {X 0,Y 327.948,Z 1015.161,A -85,B 0,C 180,E1 16471.223,E2 16471.223} C_VEL
LIN {X 0,Y 327.953,Z 1015.042,A -85,B 0,C 180,E1 16467.904,E2 16467.904} C_VEL
LIN {X 0,Y 327.951,Z 1013.43,A -85,B 0,C 180,E1 16464.051,E2 16464.051} C_VEL
LIN {X 0,Y 328.059,Z 1010.797,A -85,B 0,C 180,E1 16460.706,E2 16460.706} C_VEL
LIN {X 0,Y 328.47,Z 1006.364,A -85,B 0,C 180,E1 16456.805,E2 16456.805} C_VEL
LIN {X 0,Y 329.357,Z 1000.367,A -85,B 0,C 180,E1 16452.992,E2 16452.992} C_VEL
LIN {X 0,Y 330.99,Z 992.454,A -85,B 0,C 180,E1 16448.974,E2 16448.974} C_VEL
LIN {X 0,Y 333.244,Z 983.603,A -85,B 0,C 180,E1 16445.355,E2 16445.355} C_VEL
LIN {X 0,Y 336.663,Z 972.115,A -85,B 0,C 180,E1 16441.439,E2 16441.439} C_VEL
LIN {X 0,Y 340.566,Z 960.201,A -85,B 0,C 180,E1 16438.044,E2 16438.044} C_VEL
LIN {X 0,Y 345.469,Z 946.002,A -85,B 0,C 180,E1 16434.636,E2 16434.636} C_VEL
LIN {X 0,Y 350.826,Z 931.08,A -85,B 0,C 180,E1 16431.595,E2 16431.595} C_VEL
LIN {X 0,Y 356.601,Z 914.681,A -85,B 0,C 180,E1 16428.79,E2 16428.79} C_VEL
LIN {X 0,Y 362.729,Z 897.09,A -85,B 0,C 180,E1 16426.228,E2 16426.228} C_VEL
LIN {X 0,Y 368.619,Z 879.209,A -85,B 0,C 180,E1 16424.052,E2 16424.052} C_VEL
LIN {X 0,Y 374.745,Z 859.503,A -85,B 0,C 180,E1 16422.026,E2 16422.026} C_VEL
LIN {X 0,Y 380.101,Z 840.582,A -85,B 0,C 180,E1 16420.409,E2 16420.409} C_VEL
LIN {X 0,Y 385.691,Z 818.568,A -85,B 0,C 180,E1 16418.855,E2 16418.855} C_VEL
LIN {X 0,Y 390.114,Z 798.567,A -85,B 0,C 180,E1 16417.714,E2 16417.714} C_VEL
LIN {X 0,Y 394.512,Z 774.738,A -85,B 0,C 180,E1 16416.644,E2 16416.644} C_VEL
LIN {X 0,Y 397.832,Z 752.433,A -85,B 0,C 180,E1 16415.893,E2 16415.893} C_VEL
LIN {X 0,Y 400.143,Z 728.883,A -85,B 0,C 180,E1 16415.32,E2 16415.32} C_VEL
LIN {X 0,Y 411.562,Z 527.615,A -85,B 0,C 180,E1 16411.404,E2 16411.404} C_VEL
LIN {X 0,Y 413.517,Z 494.258,A -85,B 0,C 180,E1 16410.756,E2 16410.756} C_VEL
LIN {X 0,Y 405.695,Z 481.231,A -85,B 0,C 180,E1 16408.402,E2 16408.402} C_VEL
LIN {X 0,Y 398.988,Z 470.591,A -85,B 0,C 180,E1 16406.171,E2 16406.171} C_VEL
LIN {X 0,Y 391.714,Z 459.712,A -85,B 0,C 180,E1 16403.465,E2 16403.465} C_VEL
LIN {X 0,Y 386.851,Z 453.167,A -85,B 0,C 180,E1 16401.452,E2 16401.452} C_VEL
LIN {X 0,Y 382.825,Z 448.006,A -85,B 0,C 180,E1 16399.609,E2 16399.609} C_VEL
LIN {X 0,Y 379.155,Z 443.255,A -85,B 0,C 180,E1 16397.733,E2 16397.733} C_VEL
LIN {X 0,Y 375.3,Z 438.918,A -85,B 0,C 180,E1 16395.53,E2 16395.53} C_VEL
LIN {X 0,Y 374.069,Z 436.982,A -85,B 0,C 180,E1 16394.71,E2 16394.71} C_VEL
LIN {X 0,Y 370.835,Z 433.948,A -85,B 0,C 180,E1 16392.456,E2 16392.456} C_VEL
LIN {X 0,Y 369.122,Z 430.935,A -85,B 0,C 180,E1 16390.93,E2 16390.93} C_VEL
LIN {X 0,Y 365.683,Z 428.171,A -85,B 0,C 180,E1 16387.383,E2 16387.383} C_VEL
LIN {X 0,Y 364.158,Z 424.585,A -85,B 0,C 180,E1 16384.567,E2 16384.567} C_VEL
LIN {X 0,Y 363.289,Z 424.345,A -85,B 0,C 180,E1 16377.002,E2 16377.002} C_VEL
LIN {X 0,Y 364.293,Z 424.817,A -85,B 0,C 180,E1 16374.566,E2 16374.566} C_VEL
LIN {X 0,Y 365.733,Z 428.181,A -85,B 0,C 180,E1 16371.985,E2 16371.985} C_VEL
LIN {X 0,Y 369.01,Z 430.879,A -85,B 0,C 180,E1 16368.591,E2 16368.591} C_VEL
LIN {X 0,Y 369.682,Z 431.886,A -85,B 0,C 180,E1 16367.979,E2 16367.979} C_VEL
LIN {X 0,Y 372.228,Z 435.52,A -85,B 0,C 180,E1 16365.93,E2 16365.93} C_VEL
LIN {X 0,Y 374.553,Z 437.626,A -85,B 0,C 180,E1 16364.398,E2 16364.398} C_VEL
LIN {X 0,Y 377.631,Z 441.805,A -85,B 0,C 180,E1 16362.511,E2 16362.511} C_VEL
LIN {X 0,Y 379.395,Z 443.597,A -85,B 0,C 180,E1 16361.564,E2 16361.564} C_VEL
LIN {X 0,Y 382.948,Z 448.146,A -85,B 0,C 180,E1 16359.76,E2 16359.76} C_VEL
LIN {X 0,Y 388.541,Z 455.394,A -85,B 0,C 180,E1 16357.254,E2 16357.254} C_VEL
LIN {X 0,Y 393.297,Z 461.677,A -85,B 0,C 180,E1 16355.359,E2 16355.359} C_VEL
LIN {X 0,Y 399.277,Z 469.719,A -85,B 0,C 180,E1 16353.208,E2 16353.208} C_VEL
LIN {X 0,Y 408.096,Z 482.353,A -85,B 0,C 180,E1 16350.376,E2 16350.376} C_VEL
LIN {X 0,Y 413.428,Z 490.696,A -85,B 0,C 180,E1 16348.81,E2 16348.81} C_VEL
LIN {X 0,Y 401.585,Z 697.825,A -85,B 0,C 180,E1 16344.799,E2 16344.799} C_VEL
LIN {X 0,Y 399.519,Z 725.131,A -85,B 0,C 180,E1 16344.201,E2 16344.201} C_VEL
LIN {X 0,Y 396.823,Z 747.571,A -85,B 0,C 180,E1 16343.516,E2 16343.516} C_VEL
LIN {X 0,Y 393.219,Z 769.587,A -85,B 0,C 180,E1 16342.597,E2 16342.597} C_VEL
LIN {X 0,Y 389.069,Z 790.783,A -85,B 0,C 180,E1 16341.484,E2 16341.484} C_VEL
LIN {X 0,Y 384.221,Z 811.216,A -85,B 0,C 180,E1 16340.137,E2 16340.137} C_VEL
LIN {X 0,Y 378.869,Z 831.371,A -85,B 0,C 180,E1 16338.538,E2 16338.538} C_VEL
LIN {X 0,Y 373.296,Z 849.913,A -85,B 0,C 180,E1 16336.757,E2 16336.757} C_VEL
LIN {X 0,Y 367.214,Z 868.704,A -85,B 0,C 180,E1 16334.62,E2 16334.62} C_VEL
LIN {X 0,Y 361.486,Z 885.12,A -85,B 0,C 180,E1 16332.395,E2 16332.395} C_VEL
LIN {X 0,Y 355.359,Z 902.046,A -85,B 0,C 180,E1 16329.689,E2 16329.689} C_VEL
LIN {X 0,Y 349.831,Z 916.855,A -85,B 0,C 180,E1 16326.879,E2 16326.879} C_VEL
LIN {X 0,Y 344.277,Z 931.661,A -85,B 0,C 180,E1 16323.538,E2 16323.538} C_VEL
LIN {X 0,Y 339.772,Z 944.115,A -85,B 0,C 180,E1 16320.208,E2 16320.208} C_VEL
LIN {X 0,Y 335.813,Z 955.497,A -85,B 0,C 180,E1 16316.523,E2 16316.523} C_VEL
LIN {X 0,Y 332.693,Z 965.527,A -85,B 0,C 180,E1 16312.621,E2 16312.621} C_VEL
LIN {X 0,Y 330.668,Z 972.968,A -85,B 0,C 180,E1 16309.058,E2 16309.058} C_VEL
LIN {X 0,Y 329.17,Z 979.841,A -85,B 0,C 180,E1 16304.96,E2 16304.96} C_VEL
LIN {X 0,Y 328.453,Z 984.356,A -85,B 0,C 180,E1 16301.411,E2 16301.411} C_VEL
LIN {X 0,Y 328.072,Z 987.951,A -85,B 0,C 180,E1 16297.529,E2 16297.529} C_VEL
LIN {X 0,Y 327.973,Z 989.851,A -85,B 0,C 180,E1 16294.02,E2 16294.02} C_VEL
LIN {X 0,Y 327.951,Z 990.275,A -85,B 0,C 180,E1 16292.892,E2 16292.892} C_VEL
LIN {X 0,Y 327.095,Z 990.679,A -85,B 0,C 180,E1 16291.643,E2 16291.643} C_VEL
LIN {X 0,Y 323.413,Z 990.986,A -85,B 0,C 180,E1 16289.573,E2 16289.573} C_VEL
LIN {X 0,Y 320.304,Z 990.751,A -85,B 0,C 180,E1 16287.542,E2 16287.542} C_VEL
LIN {X 0,Y 319.957,Z 990.503,A -85,B 0,C 180,E1 16286.743,E2 16286.743} C_VEL
LIN {X 0,Y 320.054,Z 988.856,A -85,B 0,C 180,E1 16283.182,E2 16283.182} C_VEL
LIN {X 0,Y 320.34,Z 985.931,A -85,B 0,C 180,E1 16279.389,E2 16279.389} C_VEL
LIN {X 0,Y 321.086,Z 981.257,A -85,B 0,C 180,E1 16275.392,E2 16275.392} C_VEL
LIN {X 0,Y 322.463,Z 975.159,A -85,B 0,C 180,E1 16271.377,E2 16271.377} C_VEL
LIN {X 0,Y 324.536,Z 967.61,A -85,B 0,C 180,E1 16267.543,E2 16267.543} C_VEL
LIN {X 0,Y 327.508,Z 958.565,A -85,B 0,C 180,E1 16263.728,E2 16263.728} C_VEL
LIN {X 0,Y 331.445,Z 947.537,A -85,B 0,C 180,E1 16259.953,E2 16259.953} C_VEL
LIN {X 0,Y 336.434,Z 934.542,A -85,B 0,C 180,E1 16256.241,E2 16256.241} C_VEL
LIN {X 0,Y 341.556,Z 921.527,A -85,B 0,C 180,E1 16253.127,E2 16253.127} C_VEL
LIN {X 0,Y 347.49,Z 906.428,A -85,B 0,C 180,E1 16250.09,E2 16250.09} C_VEL
LIN {X 0,Y 353.429,Z 891.047,A -85,B 0,C 180,E1 16247.463,E2 16247.463} C_VEL
LIN {X 0,Y 359.747,Z 873.771,A -85,B 0,C 180,E1 16244.987,E2 16244.987} C_VEL
LIN {X 0,Y 366.214,Z 855.242,A -85,B 0,C 180,E1 16242.747,E2 16242.747} C_VEL
LIN {X 0,Y 372.129,Z 836.416,A -85,B 0,C 180,E1 16240.864,E2 16240.864} C_VEL
LIN {X 0,Y 377.9,Z 816.384,A -85,B 0,C 180,E1 16239.182,E2 16239.182} C_VEL
LIN {X 0,Y 382.845,Z 796.564,A -85,B 0,C 180,E1 16237.82,E2 16237.82} C_VEL
LIN {X 0,Y 387.438,Z 775.436,A -85,B 0,C 180,E1 16236.63,E2 16236.63} C_VEL
LIN {X 0,Y 391.051,Z 754.936,A -85,B 0,C 180,E1 16235.721,E2 16235.721} C_VEL
LIN {X 0,Y 394.213,Z 732.509,A -85,B 0,C 180,E1 16234.953,E2 16234.953} C_VEL
LIN {X 0,Y 396.295,Z 710.42,A -85,B 0,C 180,E1 16234.411,E2 16234.411} C_VEL
LIN {X 0,Y 408.625,Z 503.84,A -85,B 0,C 180,E1 16230.384,E2 16230.384} C_VEL
LIN {X 0,Y 409.098,Z 494.871,A -85,B 0,C 180,E1 16230.19,E2 16230.19} C_VEL
LIN {X 0,Y 399.767,Z 480.785,A -85,B 0,C 180,E1 16227.239,E2 16227.239} C_VEL
LIN {X 0,Y 391.723,Z 469.643,A -85,B 0,C 180,E1 16224.345,E2 16224.345} C_VEL
LIN {X 0,Y 387.848,Z 464.494,A -85,B 0,C 180,E1 16222.789,E2 16222.789} C_VEL
LIN {X 0,Y 384.699,Z 460.269,A -85,B 0,C 180,E1 16221.418,E2 16221.418} C_VEL
LIN {X 0,Y 381.079,Z 455.506,A -85,B 0,C 180,E1 16219.704,E2 16219.704} C_VEL
LIN {X 0,Y 376.965,Z 450.227,A -85,B 0,C 180,E1 16217.521,E2 16217.521} C_VEL
LIN {X 0,Y 373.538,Z 446.077,A -85,B 0,C 180,E1 16215.447,E2 16215.447} C_VEL
LIN {X 0,Y 372.555,Z 444.629,A -85,B 0,C 180,E1 16214.772,E2 16214.772} C_VEL
LIN {X 0,Y 369.274,Z 441.231,A -85,B 0,C 180,E1 16212.351,E2 16212.351} C_VEL
LIN {X 0,Y 367.972,Z 438.797,A -85,B 0,C 180,E1 16211.124,E2 16211.124} C_VEL
LIN {X 0,Y 364.663,Z 436.069,A -85,B 0,C 180,E1 16207.563,E2 16207.563} C_VEL
LIN {X 0,Y 363.168,Z 432.509,A -85,B 0,C 180,E1 16204.58,E2 16204.58} C_VEL
LIN {X 0,Y 362.777,Z 432.415,A -85,B 0,C 180,E1 16196.84,E2 16196.84} C_VEL
LIN {X 0,Y 363.286,Z 432.85,A -85,B 0,C 180,E1 16195.581,E2 16195.581} C_VEL
LIN {X 0,Y 365.246,Z 436.842,A -85,B 0,C 180,E1 16192.133,E2 16192.133} C_VEL
LIN {X 0,Y 368.224,Z 439.146,A -85,B 0,C 180,E1 16189.122,E2 16189.122} C_VEL
LIN {X 0,Y 370.599,Z 443.034,A -85,B 0,C 180,E1 16187.06,E2 16187.06} C_VEL
LIN {X 0,Y 373.119,Z 445.306,A -85,B 0,C 180,E1 16185.331,E2 16185.331} C_VEL
LIN {X 0,Y 376.305,Z 449.663,A -85,B 0,C 180,E1 16183.324,E2 16183.324} C_VEL
LIN {X 0,Y 377.822,Z 451.343,A -85,B 0,C 180,E1 16182.481,E2 16182.481} C_VEL
LIN {X 0,Y 381.69,Z 456.089,A -85,B 0,C 180,E1 16180.489,E2 16180.489} C_VEL
LIN {X 0,Y 387.028,Z 463.39,A -85,B 0,C 180,E1 16178.041,E2 16178.041} C_VEL
LIN {X 0,Y 391.856,Z 470.316,A -85,B 0,C 180,E1 16176.065,E2 16176.065} C_VEL
LIN {X 0,Y 399.891,Z 482.75,A -85,B 0,C 180,E1 16173.133,E2 16173.133} C_VEL
LIN {X 0,Y 408.788,Z 497.693,A -85,B 0,C 180,E1 16170.271,E2 16170.271} C_VEL
LIN {X 0,Y 409.239,Z 498.953,A -85,B 0,C 180,E1 16170.118,E2 16170.118} C_VEL
LIN {X 0,Y 396.615,Z 713.004,A -85,B 0,C 180,E1 16165.954,E2 16165.954} C_VEL
LIN {X 0,Y 394.394,Z 741.985,A -85,B 0,C 180,E1 16165.328,E2 16165.328} C_VEL
LIN {X 0,Y 391.518,Z 764.176,A -85,B 0,C 180,E1 16164.687,E2 16164.687} C_VEL
LIN {X 0,Y 387.677,Z 786.238,A -85,B 0,C 180,E1 16163.821,E2 16163.821} C_VEL
LIN {X 0,Y 383.416,Z 806.801,A -85,B 0,C 180,E1 16162.793,E2 16162.793} C_VEL
LIN {X 0,Y 378.259,Z 827.774,A -85,B 0,C 180,E1 16161.475,E2 16161.475} C_VEL
LIN {X 0,Y 372.632,Z 848.266,A -85,B 0,C 180,E1 16159.912,E2 16159.912} C_VEL
LIN {X 0,Y 366.456,Z 868.157,A -85,B 0,C 180,E1 16158.051,E2 16158.051} C_VEL
LIN {X 0,Y 360.089,Z 887.386,A -85,B 0,C 180,E1 16155.905,E2 16155.905} C_VEL
LIN {X 0,Y 353.898,Z 904.792,A -85,B 0,C 180,E1 16153.574,E2 16153.574} C_VEL
LIN {X 0,Y 347.237,Z 922.865,A -85,B 0,C 180,E1 16150.703,E2 16150.703} C_VEL
LIN {X 0,Y 341.689,Z 937.669,A -85,B 0,C 180,E1 16147.912,E2 16147.912} C_VEL
LIN {X 0,Y 336.179,Z 952.455,A -85,B 0,C 180,E1 16144.612,E2 16144.612} C_VEL
LIN {X 0,Y 331.59,Z 965.278,A -85,B 0,C 180,E1 16141.238,E2 16141.238} C_VEL
LIN {X 0,Y 327.699,Z 976.748,A -85,B 0,C 180,E1 16137.628,E2 16137.628} C_VEL
LIN {X 0,Y 324.623,Z 987.055,A -85,B 0,C 180,E1 16133.794,E2 16133.794} C_VEL
LIN {X 0,Y 322.458,Z 995.44,A -85,B 0,C 180,E1 16129.941,E2 16129.941} C_VEL
LIN {X 0,Y 321.032,Z 1002.646,A -85,B 0,C 180,E1 16125.906,E2 16125.906} C_VEL
LIN {X 0,Y 320.293,Z 1007.814,A -85,B 0,C 180,E1 16122.072,E2 16122.072} C_VEL
LIN {X 0,Y 320.021,Z 1011.652,A -85,B 0,C 180,E1 16118.263,E2 16118.263} C_VEL
LIN {X 0,Y 319.95,Z 1014.033,A -85,B 0,C 180,E1 16114.301,E2 16114.301} C_VEL
LIN {X 0,Y 319.949,Z 1014.884,A -85,B 0,C 180,E1 16111.075,E2 16111.075} C_VEL
LIN {X 0,Y 319.942,Z 1014.66,A -85,B 0,C 180,E1 16107.314,E2 16107.314} C_VEL
LIN {X 0,Y 319.971,Z 1012.894,A -85,B 0,C 180,E1 16103.542,E2 16103.542} C_VEL
LIN {X 0,Y 320.083,Z 1010.162,A -85,B 0,C 180,E1 16100.109,E2 16100.109} C_VEL
LIN {X 0,Y 320.623,Z 1005.224,A -85,B 0,C 180,E1 16095.892,E2 16095.892} C_VEL
LIN {X 0,Y 321.577,Z 999.547,A -85,B 0,C 180,E1 16092.262,E2 16092.262} C_VEL
LIN {X 0,Y 323.493,Z 991.149,A -85,B 0,C 180,E1 16088.008,E2 16088.008} C_VEL
LIN {X 0,Y 325.958,Z 982.347,A -85,B 0,C 180,E1 16084.377,E2 16084.377} C_VEL
LIN {X 0,Y 329.521,Z 971.193,A -85,B 0,C 180,E1 16080.555,E2 16080.555} C_VEL
LIN {X 0,Y 333.647,Z 959.429,A -85,B 0,C 180,E1 16077.157,E2 16077.157} C_VEL
LIN {X 0,Y 338.659,Z 945.685,A -85,B 0,C 180,E1 16073.814,E2 16073.814} C_VEL
LIN {X 0,Y 344.301,Z 930.763,A -85,B 0,C 180,E1 16070.729,E2 16070.729} C_VEL
LIN {X 0,Y 350.354,Z 914.365,A -85,B 0,C 180,E1 16067.889,E2 16067.889} C_VEL
LIN {X 0,Y 356.775,Z 896.775,A -85,B 0,C 180,E1 16065.305,E2 16065.305} C_VEL
LIN {X 0,Y 362.994,Z 878.66,A -85,B 0,C 180,E1 16063.086,E2 16063.086} C_VEL
LIN {X 0,Y 369.544,Z 858.289,A -85,B 0,C 180,E1 16060.994,E2 16060.994} C_VEL
LIN {X 0,Y 375.127,Z 839.24,A -85,B 0,C 180,E1 16059.372,E2 16059.372} C_VEL
LIN {X 0,Y 380.924,Z 816.963,A -85,B 0,C 180,E1 16057.817,E2 16057.817} C_VEL
LIN {X 0,Y 385.653,Z 796.169,A -85,B 0,C 180,E1 16056.648,E2 16056.648} C_VEL
LIN {X 0,Y 389.937,Z 773.227,A -85,B 0,C 180,E1 16055.644,E2 16055.644} C_VEL
LIN {X 0,Y 393.414,Z 750.179,A -85,B 0,C 180,E1 16054.887,E2 16054.887} C_VEL
LIN {X 0,Y 395.656,Z 727.057,A -85,B 0,C 180,E1 16054.336,E2 16054.336} C_VEL
LIN {X 0,Y 407.622,Z 523.979,A -85,B 0,C 180,E1 16050.372,E2 16050.372} C_VEL
LIN {X 0,Y 409.13,Z 498.43,A -85,B 0,C 180,E1 16049.863,E2 16049.863} C_VEL
LIN {X 0,Y 400.674,Z 484.138,A -85,B 0,C 180,E1 16047.172,E2 16047.172} C_VEL
LIN {X 0,Y 393.35,Z 472.637,A -85,B 0,C 180,E1 16044.557,E2 16044.557} C_VEL
LIN {X 0,Y 388.076,Z 464.847,A -85,B 0,C 180,E1 16042.455,E2 16042.455} C_VEL
LIN {X 0,Y 384.585,Z 460.169,A -85,B 0,C 180,E1 16040.945,E2 16040.945} C_VEL
LIN {X 0,Y 380.957,Z 455.402,A -85,B 0,C 180,E1 16039.231,E2 16039.231} C_VEL
LIN {X 0,Y 376.829,Z 450.151,A -85,B 0,C 180,E1 16037.049,E2 16037.049} C_VEL
LIN {X 0,Y 373.511,Z 446.094,A -85,B 0,C 180,E1 16035.05,E2 16035.05} C_VEL
LIN {X 0,Y 372.637,Z 444.711,A -85,B 0,C 180,E1 16034.45,E2 16034.45} C_VEL
LIN {X 0,Y 369.477,Z 441.636,A -85,B 0,C 180,E1 16032.185,E2 16032.185} C_VEL
LIN {X 0,Y 367.978,Z 438.822,A -85,B 0,C 180,E1 16030.806,E2 16030.806} C_VEL
LIN {X 0,Y 364.481,Z 435.89,A -85,B 0,C 180,E1 16027.091,E2 16027.091} C_VEL
LIN {X 0,Y 363.104,Z 432.513,A -85,B 0,C 180,E1 16024.422,E2 16024.422} C_VEL
LIN {X 0,Y 362.315,Z 432.287,A -85,B 0,C 180,E1 16016.994,E2 16016.994} C_VEL
LIN {X 0,Y 363.235,Z 432.746,A -85,B 0,C 180,E1 16014.709,E2 16014.709} C_VEL
LIN {X 0,Y 364.641,Z 436.063,A -85,B 0,C 180,E1 16012.12,E2 16012.12} C_VEL
LIN {X 0,Y 367.96,Z 438.806,A -85,B 0,C 180,E1 16008.638,E2 16008.638} C_VEL
LIN {X 0,Y 370.529,Z 442.903,A -85,B 0,C 180,E1 16006.422,E2 16006.422} C_VEL
LIN {X 0,Y 373.057,Z 445.295,A -85,B 0,C 180,E1 16004.692,E2 16004.692} C_VEL
LIN {X 0,Y 376.274,Z 449.622,A -85,B 0,C 180,E1 16002.685,E2 16002.685} C_VEL
LIN {X 0,Y 377.866,Z 451.405,A -85,B 0,C 180,E1 16001.806,E2 16001.806} C_VEL
LIN {X 0,Y 382.483,Z 457.408,A -85,B 0,C 180,E1 15999.455,E2 15999.455} C_VEL
LIN {X 0,Y 386.647,Z 462.897,A -85,B 0,C 180,E1 15997.577,E2 15997.577} C_VEL
LIN {X 0,Y 391.42,Z 469.3,A -85,B 0,C 180,E1 15995.635,E2 15995.635} C_VEL
LIN {X 0,Y 397.506,Z 477.76,A -85,B 0,C 180,E1 15993.402,E2 15993.402} C_VEL
LIN {X 0,Y 405.421,Z 489.282,A -85,B 0,C 180,E1 15990.806,E2 15990.806} C_VEL
LIN {X 0,Y 409.084,Z 495.171,A -85,B 0,C 180,E1 15989.687,E2 15989.687} C_VEL
LIN {X 0,Y 396.768,Z 702.721,A -85,B 0,C 180,E1 15985.653,E2 15985.653} C_VEL
LIN {X 0,Y 394.748,Z 726.807,A -85,B 0,C 180,E1 15985.106,E2 15985.106} C_VEL
LIN {X 0,Y 391.862,Z 749.571,A -85,B 0,C 180,E1 15984.395,E2 15984.395} C_VEL
LIN {X 0,Y 388.196,Z 770.951,A -85,B 0,C 180,E1 15983.489,E2 15983.489} C_VEL
LIN {X 0,Y 383.829,Z 792.22,A -85,B 0,C 180,E1 15982.355,E2 15982.355} C_VEL
LIN {X 0,Y 379.084,Z 811.526,A -85,B 0,C 180,E1 15981.076,E2 15981.076} C_VEL
LIN {X 0,Y 373.542,Z 831.681,A -85,B 0,C 180,E1 15979.472,E2 15979.472} C_VEL
LIN {X 0,Y 367.761,Z 850.224,A -85,B 0,C 180,E1 15977.681,E2 15977.681} C_VEL
LIN {X 0,Y 361.44,Z 869.015,A -85,B 0,C 180,E1 15975.53,E2 15975.53} C_VEL
LIN {X 0,Y 355.552,Z 885.204,A -85,B 0,C 180,E1 15973.32,E2 15973.32} C_VEL
LIN {X 0,Y 349.053,Z 902.359,A -85,B 0,C 180,E1 15970.553,E2 15970.553} C_VEL
LIN {X 0,Y 343.26,Z 917.168,A -85,B 0,C 180,E1 15967.706,E2 15967.706} C_VEL
LIN {X 0,Y 337.607,Z 931.467,A -85,B 0,C 180,E1 15964.443,E2 15964.443} C_VEL
LIN {X 0,Y 332.873,Z 943.805,A -85,B 0,C 180,E1 15961.103,E2 15961.103} C_VEL
LIN {X 0,Y 328.615,Z 955.307,A -85,B 0,C 180,E1 15957.347,E2 15957.347} C_VEL
LIN {X 0,Y 325.37,Z 965.05,A -85,B 0,C 180,E1 15953.543,E2 15953.543} C_VEL
LIN {X 0,Y 323.019,Z 972.933,A -85,B 0,C 180,E1 15949.715,E2 15949.715} C_VEL
LIN {X 0,Y 321.412,Z 979.655,A -85,B 0,C 180,E1 15945.7,E2 15945.7} C_VEL
LIN {X 0,Y 320.537,Z 984.461,A -85,B 0,C 180,E1 15941.879,E2 15941.879} C_VEL
LIN {X 0,Y 320.113,Z 988.143,A -85,B 0,C 180,E1 15937.898,E2 15937.898} C_VEL
LIN {X 0,Y 319.983,Z 990.151,A -85,B 0,C 180,E1 15934.12,E2 15934.12} C_VEL
LIN {X 0,Y 319.946,Z 990.93,A -85,B 0,C 180,E1 15930.716,E2 15930.716} C_VEL
LIN {X 0,Y 319.956,Z 990.515,A -85,B 0,C 180,E1 15926.775,E2 15926.775} C_VEL
LIN {X 0,Y 319.957,Z 990.503,A -85,B 0,C 180,E1 15926.743,E2 15926.743} C_VEL
LIN {X 0,Y 318.988,Z 990.051,A -85,B 0,C 180,E1 15925.366,E2 15925.366} C_VEL
LIN {X 0,Y 314.813,Z 989.015,A -85,B 0,C 180,E1 15922.955,E2 15922.955} C_VEL
LIN {X 0,Y 312.476,Z 987.923,A -85,B 0,C 180,E1 15921.17,E2 15921.17} C_VEL
LIN {X 0,Y 312.256,Z 987.346,A -85,B 0,C 180,E1 15920.46,E2 15920.46} C_VEL
LIN {X 0,Y 312.853,Z 983.47,A -85,B 0,C 180,E1 15916.509,E2 15916.509} C_VEL
LIN {X 0,Y 314.069,Z 977.819,A -85,B 0,C 180,E1 15912.397,E2 15912.397} C_VEL
LIN {X 0,Y 316.105,Z 970.667,A -85,B 0,C 180,E1 15908.282,E2 15908.282} C_VEL
LIN {X 0,Y 318.946,Z 962.027,A -85,B 0,C 180,E1 15904.369,E2 15904.369} C_VEL
LIN {X 0,Y 322.799,Z 951.77,A -85,B 0,C 180,E1 15900.498,E2 15900.498} C_VEL
LIN {X 0,Y 327.434,Z 940.057,A -85,B 0,C 180,E1 15896.87,E2 15896.87} C_VEL
LIN {X 0,Y 333.396,Z 925.618,A -85,B 0,C 180,E1 15893.149,E2 15893.149} C_VEL
LIN {X 0,Y 339.402,Z 911.216,A -85,B 0,C 180,E1 15890.048,E2 15890.048} C_VEL
LIN {X 0,Y 345.803,Z 895.348,A -85,B 0,C 180,E1 15887.202,E2 15887.202} C_VEL
LIN {X 0,Y 352.345,Z 878.668,A -85,B 0,C 180,E1 15884.661,E2 15884.661} C_VEL
LIN {X 0,Y 358.816,Z 860.823,A -85,B 0,C 180,E1 15882.404,E2 15882.404} C_VEL
LIN {X 0,Y 365.355,Z 841.539,A -85,B 0,C 180,E1 15880.352,E2 15880.352} C_VEL
LIN {X 0,Y 371.086,Z 822.68,A -85,B 0,C 180,E1 15878.69,E2 15878.69} C_VEL
LIN {X 0,Y 376.857,Z 801.348,A -85,B 0,C 180,E1 15877.138,E2 15877.138} C_VEL
LIN {X 0,Y 381.296,Z 782.196,A -85,B 0,C 180,E1 15876,E2 15876} C_VEL
LIN {X 0,Y 385.829,Z 758.788,A -85,B 0,C 180,E1 15874.896,E2 15874.896} C_VEL
LIN {X 0,Y 388.955,Z 738.192,A -85,B 0,C 180,E1 15874.15,E2 15874.15} C_VEL
LIN {X 0,Y 391.56,Z 714.116,A -85,B 0,C 180,E1 15873.519,E2 15873.519} C_VEL
LIN {X 0,Y 403.848,Z 516.427,A -85,B 0,C 180,E1 15869.645,E2 15869.645} C_VEL
LIN {X 0,Y 404.901,Z 499.476,A -85,B 0,C 180,E1 15869.308,E2 15869.308} C_VEL
LIN {X 0,Y 396.919,Z 487.293,A -85,B 0,C 180,E1 15866.681,E2 15866.681} C_VEL
LIN {X 0,Y 389.418,Z 476.669,A -85,B 0,C 180,E1 15863.894,E2 15863.894} C_VEL
LIN {X 0,Y 383.414,Z 468.35,A -85,B 0,C 180,E1 15861.333,E2 15861.333} C_VEL
LIN {X 0,Y 379.087,Z 462.749,A -85,B 0,C 180,E1 15859.25,E2 15859.25} C_VEL
LIN {X 0,Y 375.342,Z 457.803,A -85,B 0,C 180,E1 15857.199,E2 15857.199} C_VEL
LIN {X 0,Y 371.995,Z 453.628,A -85,B 0,C 180,E1 15855.113,E2 15855.113} C_VEL
LIN {X 0,Y 371.141,Z 452.35,A -85,B 0,C 180,E1 15854.51,E2 15854.51} C_VEL
LIN {X 0,Y 367.851,Z 448.782,A -85,B 0,C 180,E1 15852.002,E2 15852.002} C_VEL
LIN {X 0,Y 366.66,Z 446.596,A -85,B 0,C 180,E1 15850.846,E2 15850.846} C_VEL
LIN {X 0,Y 363.472,Z 443.797,A -85,B 0,C 180,E1 15847.27,E2 15847.27} C_VEL
LIN {X 0,Y 362.123,Z 440.437,A -85,B 0,C 180,E1 15844.434,E2 15844.434} C_VEL
LIN {X 0,Y 361.862,Z 440.376,A -85,B 0,C 180,E1 15836.674,E2 15836.674} C_VEL
LIN {X 0,Y 362.236,Z 440.777,A -85,B 0,C 180,E1 15835.726,E2 15835.726} C_VEL
LIN {X 0,Y 364.272,Z 444.85,A -85,B 0,C 180,E1 15832.112,E2 15832.112} C_VEL
LIN {X 0,Y 366.984,Z 447.048,A -85,B 0,C 180,E1 15829.324,E2 15829.324} C_VEL
LIN {X 0,Y 369.525,Z 451.05,A -85,B 0,C 180,E1 15827.102,E2 15827.102} C_VEL
LIN {X 0,Y 371.687,Z 453.06,A -85,B 0,C 180,E1 15825.592,E2 15825.592} C_VEL
LIN {X 0,Y 374.952,Z 457.474,A -85,B 0,C 180,E1 15823.502,E2 15823.502} C_VEL
LIN {X 0,Y 376.367,Z 459.226,A -85,B 0,C 180,E1 15822.691,E2 15822.691} C_VEL
LIN {X 0,Y 380.683,Z 464.799,A -85,B 0,C 180,E1 15820.435,E2 15820.435} C_VEL
LIN {X 0,Y 384.904,Z 470.529,A -85,B 0,C 180,E1 15818.474,E2 15818.474} C_VEL
LIN {X 0,Y 389.715,Z 477.608,A -85,B 0,C 180,E1 15816.448,E2 15816.448} C_VEL
LIN {X 0,Y 397.421,Z 489.803,A -85,B 0,C 180,E1 15813.557,E2 15813.557} C_VEL
LIN {X 0,Y 405.025,Z 502.793,A -85,B 0,C 180,E1 15811.025,E2 15811.025} C_VEL
LIN {X 0,Y 391.967,Z 716.101,A -85,B 0,C 180,E1 15806.862,E2 15806.862} C_VEL
LIN {X 0,Y 389.779,Z 742.512,A -85,B 0,C 180,E1 15806.28,E2 15806.28} C_VEL
LIN {X 0,Y 386.689,Z 765.424,A -85,B 0,C 180,E1 15805.612,E2 15805.612} C_VEL
LIN {X 0,Y 382.632,Z 787.555,A -85,B 0,C 180,E1 15804.726,E2 15804.726} C_VEL
LIN {X 0,Y 378.013,Z 808.845,A -85,B 0,C 180,E1 15803.642,E2 15803.642} C_VEL
LIN {X 0,Y 372.674,Z 829.497,A -85,B 0,C 180,E1 15802.315,E2 15802.315} C_VEL
LIN {X 0,Y 366.789,Z 849.897,A -85,B 0,C 180,E1 15800.723,E2 15800.723} C_VEL
LIN {X 0,Y 360.684,Z 868.785,A -85,B 0,C 180,E1 15798.93,E2 15798.93} C_VEL
LIN {X 0,Y 353.824,Z 888.527,A -85,B 0,C 180,E1 15796.684,E2 15796.684} C_VEL
LIN {X 0,Y 347.492,Z 905.607,A -85,B 0,C 180,E1 15794.357,E2 15794.357} C_VEL
LIN {X 0,Y 340.567,Z 923.494,A -85,B 0,C 180,E1 15791.45,E2 15791.45} C_VEL
LIN {X 0,Y 334.462,Z 939.078,A -85,B 0,C 180,E1 15788.443,E2 15788.443} C_VEL
LIN {X 0,Y 328.745,Z 953.57,A -85,B 0,C 180,E1 15785.084,E2 15785.084} C_VEL
LIN {X 0,Y 323.763,Z 966.808,A -85,B 0,C 180,E1 15781.457,E2 15781.457} C_VEL
LIN {X 0,Y 319.767,Z 978.023,A -85,B 0,C 180,E1 15777.763,E2 15777.763} C_VEL
LIN {X 0,Y 316.368,Z 988.838,A -85,B 0,C 180,E1 15773.464,E2 15773.464} C_VEL
LIN {X 0,Y 314.259,Z 996.947,A -85,B 0,C 180,E1 15769.514,E2 15769.514} C_VEL
LIN {X 0,Y 312.884,Z 1003.653,A -85,B 0,C 180,E1 15765.38,E2 15765.38} C_VEL
LIN {X 0,Y 312.26,Z 1008.15,A -85,B 0,C 180,E1 15761.824,E2 15761.824} C_VEL
LIN {X 0,Y 311.984,Z 1011.884,A -85,B 0,C 180,E1 15757.735,E2 15757.735} C_VEL
LIN {X 0,Y 311.953,Z 1013.804,A -85,B 0,C 180,E1 15754.228,E2 15754.228} C_VEL
LIN {X 0,Y 311.948,Z 1014.631,A -85,B 0,C 180,E1 15750.735,E2 15750.735} C_VEL
LIN {X 0,Y 311.938,Z 1014.225,A -85,B 0,C 180,E1 15746.877,E2 15746.877} C_VEL
LIN {X 0,Y 311.969,Z 1012.591,A -85,B 0,C 180,E1 15743.376,E2 15743.376} C_VEL
LIN {X 0,Y 312.087,Z 1010.023,A -85,B 0,C 180,E1 15740.039,E2 15740.039} C_VEL
LIN {X 0,Y 312.613,Z 1005.487,A -85,B 0,C 180,E1 15735.934,E2 15735.934} C_VEL
LIN {X 0,Y 313.595,Z 999.862,A -85,B 0,C 180,E1 15732.179,E2 15732.179} C_VEL
LIN {X 0,Y 315.452,Z 992.156,A -85,B 0,C 180,E1 15728.04,E2 15728.04} C_VEL
LIN {X 0,Y 318.135,Z 982.974,A -85,B 0,C 180,E1 15724.1,E2 15724.1} C_VEL
LIN {X 0,Y 322.036,Z 971.483,A -85,B 0,C 180,E1 15720.013,E2 15720.013} C_VEL
LIN {X 0,Y 326.369,Z 959.761,A -85,B 0,C 180,E1 15716.539,E2 15716.539} C_VEL
LIN {X 0,Y 331.927,Z 945.368,A -85,B 0,C 180,E1 15712.96,E2 15712.96} C_VEL
LIN {X 0,Y 338.04,Z 929.992,A -85,B 0,C 180,E1 15709.739,E2 15709.739} C_VEL
LIN {X 0,Y 344.305,Z 913.79,A -85,B 0,C 180,E1 15706.915,E2 15706.915} C_VEL
LIN {X 0,Y 350.919,Z 896.46,A -85,B 0,C 180,E1 15704.351,E2 15704.351} C_VEL
LIN {X 0,Y 357.308,Z 878.581,A -85,B 0,C 180,E1 15702.144,E2 15702.144} C_VEL
LIN {X 0,Y 363.942,Z 858.794,A -85,B 0,C 180,E1 15700.091,E2 15700.091} C_VEL
LIN {X 0,Y 369.712,Z 839.839,A -85,B 0,C 180,E1 15698.463,E2 15698.463} C_VEL
LIN {X 0,Y 375.784,Z 817.456,A -85,B 0,C 180,E1 15696.885,E2 15696.885} C_VEL
LIN {X 0,Y 380.571,Z 797.148,A -85,B 0,C 180,E1 15695.735,E2 15695.735} C_VEL
LIN {X 0,Y 385.135,Z 773.785,A -85,B 0,C 180,E1 15694.701,E2 15694.701} C_VEL
LIN {X 0,Y 388.758,Z 750.767,A -85,B 0,C 180,E1 15693.938,E2 15693.938} C_VEL
LIN {X 0,Y 391.139,Z 727.165,A -85,B 0,C 180,E1 15693.372,E2 15693.372} C_VEL
LIN {X 0,Y 403.547,Z 524.615,A -85,B 0,C 180,E1 15689.404,E2 15689.404} C_VEL
LIN {X 0,Y 404.853,Z 502.535,A -85,B 0,C 180,E1 15688.95,E2 15688.95} C_VEL
LIN {X 0,Y 396.003,Z 487.589,A -85,B 0,C 180,E1 15685.98,E2 15685.98} C_VEL
LIN {X 0,Y 388.171,Z 475.216,A -85,B 0,C 180,E1 15682.969,E2 15682.969} C_VEL
LIN {X 0,Y 382.82,Z 467.716,A -85,B 0,C 180,E1 15680.646,E2 15680.646} C_VEL
LIN {X 0,Y 379.107,Z 462.794,A -85,B 0,C 180,E1 15678.849,E2 15678.849} C_VEL
LIN {X 0,Y 375.069,Z 457.604,A -85,B 0,C 180,E1 15676.652,E2 15676.652} C_VEL
LIN {X 0,Y 371.748,Z 453.264,A -85,B 0,C 180,E1 15674.565,E2 15674.565} C_VEL
LIN {X 0,Y 370.757,Z 452.118,A -85,B 0,C 180,E1 15673.887,E2 15673.887} C_VEL
LIN {X 0,Y 367.777,Z 448.758,A -85,B 0,C 180,E1 15671.606,E2 15671.606} C_VEL
LIN {X 0,Y 366.656,Z 446.628,A -85,B 0,C 180,E1 15670.527,E2 15670.527} C_VEL
LIN {X 0,Y 363.188,Z 443.435,A -85,B 0,C 180,E1 15666.639,E2 15666.639} C_VEL
LIN {X 0,Y 362.053,Z 440.441,A -85,B 0,C 180,E1 15664.276,E2 15664.276} C_VEL
LIN {X 0,Y 361.388,Z 440.249,A -85,B 0,C 180,E1 15656.828,E2 15656.828} C_VEL
LIN {X 0,Y 362.181,Z 440.669,A -85,B 0,C 180,E1 15654.852,E2 15654.852} C_VEL
LIN {X 0,Y 363.665,Z 444.095,A -85,B 0,C 180,E1 15652.098,E2 15652.098} C_VEL
LIN {X 0,Y 366.88,Z 446.978,A -85,B 0,C 180,E1 15648.684,E2 15648.684} C_VEL
LIN {X 0,Y 369.458,Z 450.917,A -85,B 0,C 180,E1 15646.461,E2 15646.461} C_VEL
LIN {X 0,Y 371.624,Z 453.049,A -85,B 0,C 180,E1 15644.951,E2 15644.951} C_VEL
LIN {X 0,Y 374.92,Z 457.435,A -85,B 0,C 180,E1 15642.861,E2 15642.861} C_VEL
LIN {X 0,Y 376.346,Z 459.192,A -85,B 0,C 180,E1 15642.05,E2 15642.05} C_VEL
LIN {X 0,Y 380.678,Z 464.889,A -85,B 0,C 180,E1 15639.794,E2 15639.794} C_VEL
LIN {X 0,Y 384.846,Z 470.509,A -85,B 0,C 180,E1 15637.869,E2 15637.869} C_VEL
LIN {X 0,Y 390.888,Z 478.637,A -85,B 0,C 180,E1 15635.398,E2 15635.398} C_VEL
LIN {X 0,Y 400.131,Z 492.126,A -85,B 0,C 180,E1 15632.101,E2 15632.101} C_VEL
LIN {X 0,Y 404.839,Z 499.629,A -85,B 0,C 180,E1 15630.584,E2 15630.584} C_VEL
LIN {X 0,Y 392.042,Z 707.05,A -85,B 0,C 180,E1 15626.536,E2 15626.536} C_VEL
LIN {X 0,Y 389.98,Z 729.375,A -85,B 0,C 180,E1 15626.009,E2 15626.009} C_VEL
LIN {X 0,Y 386.724,Z 753.013,A -85,B 0,C 180,E1 15625.236,E2 15625.236} C_VEL
LIN {X 0,Y 383.14,Z 773.004,A -85,B 0,C 180,E1 15624.371,E2 15624.371} C_VEL
LIN {X 0,Y 378.159,Z 795.781,A -85,B 0,C 180,E1 15623.116,E2 15623.116} C_VEL
LIN {X 0,Y 373.271,Z 814.826,A -85,B 0,C 180,E1 15621.821,E2 15621.821} C_VEL
LIN {X 0,Y 367.292,Z 835.204,A -85,B 0,C 180,E1 15620.137,E2 15620.137} C_VEL
LIN {X 0,Y 361.368,Z 853.441,A -85,B 0,C 180,E1 15618.328,E2 15618.328} C_VEL
LIN {X 0,Y 354.636,Z 872.28,A -85,B 0,C 180,E1 15616.086,E2 15616.086} C_VEL
LIN {X 0,Y 347.975,Z 889.889,A -85,B 0,C 180,E1 15613.592,E2 15613.592} C_VEL
LIN {X 0,Y 341.711,Z 905.405,A -85,B 0,C 180,E1 15610.946,E2 15610.946} C_VEL
LIN {X 0,Y 335.444,Z 920.724,A -85,B 0,C 180,E1 15607.875,E2 15607.875} C_VEL
LIN {X 0,Y 329.964,Z 933.841,A -85,B 0,C 180,E1 15604.723,E2 15604.723} C_VEL
LIN {X 0,Y 324.629,Z 947.021,A -85,B 0,C 180,E1 15600.95,E2 15600.95} C_VEL
LIN {X 0,Y 320.512,Z 957.753,A -85,B 0,C 180,E1 15597.242,E2 15597.242} C_VEL
LIN {X 0,Y 317.133,Z 967.33,A -85,B 0,C 180,E1 15593.207,E2 15593.207} C_VEL
LIN {X 0,Y 314.742,Z 975.302,A -85,B 0,C 180,E1 15589.096,E2 15589.096} C_VEL
LIN {X 0,Y 313.222,Z 981.439,A -85,B 0,C 180,E1 15584.983,E2 15584.983} C_VEL
LIN {X 0,Y 312.405,Z 986.153,A -85,B 0,C 180,E1 15580.883,E2 15580.883} C_VEL
LIN {X 0,Y 312.068,Z 989.101,A -85,B 0,C 180,E1 15576.992,E2 15576.992} C_VEL
LIN {X 0,Y 311.968,Z 990.715,A -85,B 0,C 180,E1 15573.49,E2 15573.49} C_VEL
LIN {X 0,Y 311.955,Z 991.286,A -85,B 0,C 180,E1 15569.632,E2 15569.632} C_VEL
LIN {X 0,Y 311.983,Z 990.551,A -85,B 0,C 180,E1 15565.957,E2 15565.957} C_VEL
LIN {X 0,Y 312.084,Z 988.83,A -85,B 0,C 180,E1 15562.452,E2 15562.452} C_VEL
LIN {X 0,Y 312.256,Z 987.346,A -85,B 0,C 180,E1 15560.46,E2 15560.46} C_VEL
LIN {X 0,Y 311.401,Z 986.254,A -85,B 0,C 180,E1 15559.059,E2 15559.059} C_VEL
LIN {X 0,Y 305.794,Z 982.563,A -85,B 0,C 180,E1 15555.194,E2 15555.194} C_VEL
LIN {X 0,Y 305.492,Z 981.166,A -85,B 0,C 180,E1 15554.073,E2 15554.073} C_VEL
LIN {X 0,Y 307.42,Z 974.18,A -85,B 0,C 180,E1 15549.505,E2 15549.505} C_VEL
LIN {X 0,Y 309.941,Z 966.648,A -85,B 0,C 180,E1 15545.614,E2 15545.614} C_VEL
LIN {X 0,Y 313.728,Z 956.667,A -85,B 0,C 180,E1 15541.445,E2 15541.445} C_VEL
LIN {X 0,Y 318.26,Z 945.808,A -85,B 0,C 180,E1 15537.683,E2 15537.683} C_VEL
LIN {X 0,Y 323.677,Z 933.097,A -85,B 0,C 180,E1 15534.065,E2 15534.065} C_VEL
LIN {X 0,Y 329.869,Z 919.004,A -85,B 0,C 180,E1 15530.696,E2 15530.696} C_VEL
LIN {X 0,Y 336.163,Z 904.305,A -85,B 0,C 180,E1 15527.768,E2 15527.768} C_VEL
LIN {X 0,Y 343.65,Z 886.314,A -85,B 0,C 180,E1 15524.777,E2 15524.777} C_VEL
LIN {X 0,Y 350.259,Z 869.568,A -85,B 0,C 180,E1 15522.452,E2 15522.452} C_VEL
LIN {X 0,Y 357.052,Z 850.83,A -85,B 0,C 180,E1 15520.283,E2 15520.283} C_VEL
LIN {X 0,Y 363.562,Z 831.38,A -85,B 0,C 180,E1 15518.398,E2 15518.398} C_VEL
LIN {X 0,Y 369.511,Z 810.997,A -85,B 0,C 180,E1 15516.788,E2 15516.788} C_VEL
LIN {X 0,Y 374.874,Z 790.275,A -85,B 0,C 180,E1 15515.439,E2 15515.439} C_VEL
LIN {X 0,Y 379.475,Z 768.735,A -85,B 0,C 180,E1 15514.323,E2 15514.323} C_VEL
LIN {X 0,Y 383.645,Z 744.419,A -85,B 0,C 180,E1 15513.353,E2 15513.353} C_VEL
LIN {X 0,Y 386.485,Z 722.234,A -85,B 0,C 180,E1 15512.709,E2 15512.709} C_VEL
LIN {X 0,Y 389.051,Z 687.123,A -85,B 0,C 180,E1 15511.981,E2 15511.981} C_VEL
LIN {X 0,Y 400.768,Z 504.063,A -85,B 0,C 180,E1 15508.397,E2 15508.397} C_VEL
LIN {X 0,Y 393.919,Z 493.523,A -85,B 0,C 180,E1 15506.047,E2 15506.047} C_VEL
LIN {X 0,Y 386.968,Z 483.457,A -85,B 0,C 180,E1 15503.367,E2 15503.367} C_VEL
LIN {X 0,Y 381.033,Z 475.184,A -85,B 0,C 180,E1 15500.748,E2 15500.748} C_VEL
LIN {X 0,Y 377.262,Z 470.139,A -85,B 0,C 180,E1 15498.865,E2 15498.865} C_VEL
LIN {X 0,Y 373.73,Z 465.376,A -85,B 0,C 180,E1 15496.875,E2 15496.875} C_VEL
LIN {X 0,Y 370.362,Z 460.993,A -85,B 0,C 180,E1 15494.701,E2 15494.701} C_VEL
LIN {X 0,Y 369.297,Z 459.717,A -85,B 0,C 180,E1 15493.944,E2 15493.944} C_VEL
LIN {X 0,Y 366.28,Z 456.04,A -85,B 0,C 180,E1 15491.495,E2 15491.495} C_VEL
LIN {X 0,Y 365.356,Z 454.391,A -85,B 0,C 180,E1 15490.566,E2 15490.566} C_VEL
LIN {X 0,Y 362.195,Z 451.362,A -85,B 0,C 180,E1 15486.818,E2 15486.818} C_VEL
LIN {X 0,Y 361.08,Z 448.365,A -85,B 0,C 180,E1 15484.288,E2 15484.288} C_VEL
LIN {X 0,Y 360.889,Z 448.318,A -85,B 0,C 180,E1 15476.665,E2 15476.665} C_VEL
LIN {X 0,Y 361.213,Z 448.81,A -85,B 0,C 180,E1 15475.794,E2 15475.794} C_VEL
LIN {X 0,Y 363.174,Z 452.727,A -85,B 0,C 180,E1 15472.247,E2 15472.247} C_VEL
LIN {X 0,Y 365.751,Z 454.937,A -85,B 0,C 180,E1 15469.526,E2 15469.526} C_VEL
LIN {X 0,Y 368.353,Z 458.952,A -85,B 0,C 180,E1 15467.219,E2 15467.219} C_VEL
LIN {X 0,Y 370.264,Z 460.804,A -85,B 0,C 180,E1 15465.855,E2 15465.855} C_VEL
LIN {X 0,Y 373.602,Z 465.284,A -85,B 0,C 180,E1 15463.68,E2 15463.68} C_VEL
LIN {X 0,Y 378.822,Z 472.164,A -85,B 0,C 180,E1 15460.816,E2 15460.816} C_VEL
LIN {X 0,Y 383.192,Z 478.245,A -85,B 0,C 180,E1 15458.735,E2 15458.735} C_VEL
LIN {X 0,Y 387.846,Z 485.302,A -85,B 0,C 180,E1 15456.73,E2 15456.73} C_VEL
LIN {X 0,Y 394.973,Z 496.852,A -85,B 0,C 180,E1 15453.987,E2 15453.987} C_VEL
LIN {X 0,Y 400.871,Z 507.229,A -85,B 0,C 180,E1 15451.941,E2 15451.941} C_VEL
LIN {X 0,Y 387.454,Z 718.63,A -85,B 0,C 180,E1 15447.803,E2 15447.803} C_VEL
LIN {X 0,Y 385.274,Z 743.039,A -85,B 0,C 180,E1 15447.254,E2 15447.254} C_VEL
LIN {X 0,Y 382.013,Z 766.131,A -85,B 0,C 180,E1 15446.574,E2 15446.574} C_VEL
LIN {X 0,Y 378.042,Z 787.136,A -85,B 0,C 180,E1 15445.733,E2 15445.733} C_VEL
LIN {X 0,Y 373.261,Z 808.519,A -85,B 0,C 180,E1 15444.648,E2 15444.648} C_VEL
LIN {X 0,Y 367.742,Z 829.197,A -85,B 0,C 180,E1 15443.321,E2 15443.321} C_VEL
LIN {X 0,Y 361.653,Z 849.594,A -85,B 0,C 180,E1 15441.729,E2 15441.729} C_VEL
LIN {X 0,Y 355.329,Z 868.463,A -85,B 0,C 180,E1 15439.934,E2 15439.934} C_VEL
LIN {X 0,Y 348.071,Z 888.514,A -85,B 0,C 180,E1 15437.64,E2 15437.64} C_VEL
LIN {X 0,Y 341.365,Z 905.86,A -85,B 0,C 180,E1 15435.252,E2 15435.252} C_VEL
LIN {X 0,Y 334.3,Z 923.306,A -85,B 0,C 180,E1 15432.376,E2 15432.376} C_VEL
LIN {X 0,Y 327.935,Z 938.764,A -85,B 0,C 180,E1 15429.355,E2 15429.355} C_VEL
LIN {X 0,Y 321.915,Z 953.257,A -85,B 0,C 180,E1 15425.942,E2 15425.942} C_VEL
LIN {X 0,Y 316.625,Z 966.495,A -85,B 0,C 180,E1 15422.251,E2 15422.251} C_VEL
LIN {X 0,Y 312.386,Z 977.703,A -85,B 0,C 180,E1 15418.481,E2 15418.481} C_VEL
LIN {X 0,Y 308.705,Z 988.641,A -85,B 0,C 180,E1 15414.027,E2 15414.027} C_VEL
LIN {X 0,Y 306.462,Z 996.671,A -85,B 0,C 180,E1 15410.013,E2 15410.013} C_VEL
LIN {X 0,Y 304.983,Z 1003.346,A -85,B 0,C 180,E1 15405.788,E2 15405.788} C_VEL
LIN {X 0,Y 304.272,Z 1008.059,A -85,B 0,C 180,E1 15401.947,E2 15401.947} C_VEL
LIN {X 0,Y 303.988,Z 1011.7,A -85,B 0,C 180,E1 15397.75,E2 15397.75} C_VEL
LIN {X 0,Y 303.957,Z 1013.574,A -85,B 0,C 180,E1 15394.15,E2 15394.15} C_VEL
LIN {X 0,Y 303.955,Z 1014.354,A -85,B 0,C 180,E1 15390.566,E2 15390.566} C_VEL
LIN {X 0,Y 303.944,Z 1013.854,A -85,B 0,C 180,E1 15386.606,E2 15386.606} C_VEL
LIN {X 0,Y 303.962,Z 1012.17,A -85,B 0,C 180,E1 15383.011,E2 15383.011} C_VEL
LIN {X 0,Y 304.137,Z 1009.387,A -85,B 0,C 180,E1 15379.393,E2 15379.393} C_VEL
LIN {X 0,Y 304.751,Z 1004.654,A -85,B 0,C 180,E1 15375.175,E2 15375.175} C_VEL
LIN {X 0,Y 305.893,Z 998.926,A -85,B 0,C 180,E1 15371.32,E2 15371.32} C_VEL
LIN {X 0,Y 308.122,Z 990.596,A -85,B 0,C 180,E1 15366.884,E2 15366.884} C_VEL
LIN {X 0,Y 310.984,Z 981.719,A -85,B 0,C 180,E1 15363.046,E2 15363.046} C_VEL
LIN {X 0,Y 315.246,Z 969.995,A -85,B 0,C 180,E1 15358.874,E2 15358.874} C_VEL
